KUKA KRL program: EPS_2_25618_SANMH07_A_20250918115512.src

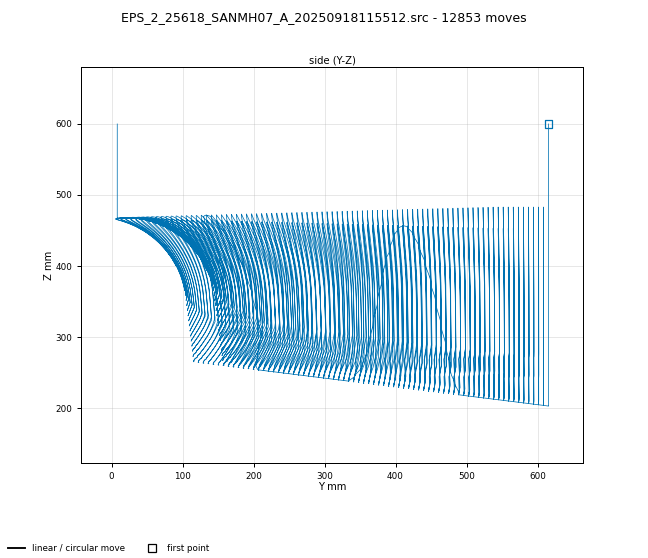
[picture p0: tool path of EPS_2_25618_SANMH07_A_20250918115512.src, 12853 of 12855 moves have a stored position in this frame; points joined in program order, loops and branches not executed]
&ACCESS RVP
&REL 4
&COMMENT QRS 19112012
&PARAM EDITMASK = *
DEF PART()
EXT BAS (BAS_COMMAND :IN,REAL :IN )
INT I
BAS (#INITMOV,0 )

;KUKA QRS Post kuka4.cps  Date:22-06-2017 !

File_ID=2844

QRS_PRE_INIT()

;Init var - Until changes are made in qrs_pre_init
Outlet_Square_prg=0
Inlet_1_Square_prg=0
Inlet_2_Square_prg=0
Inlet_3_Square_prg=0
Inlet_4_Square_prg=0
Inlet_5_Square_prg=0

Outlet_1={X 0.000, Y 540.910, Z 382.500, B 0.000, E1 0.000 }
Inlet_1={X 0.000, Y 543.050, Z 352.500, B 0.000, E1 174.000 }
Outlet_1_type=201
Inlet_1_type=201
;QRS#1=Sidecore dimensions
;QRS#2=200-8" PVC SDR 35
;QRS#3=200-8" PVC SDR 35
;QRS#4=
;QRS#5=
;QRS#6=
;QRS#7=
;QRS#8=
;QRS#9=12-08 PSX
;QRS#10=12-08 PSX
;QRS#11=
;QRS#12=
;QRS#13=
;QRS#14=
;QRS#15=
;QRS#16=1220x127x762 2,5'
;QRS#17=EPS Height
;QRS#18=483
;QRS#19=*
;QRS#20= UPDATED VERSION 22-06-2017
;QRS#21=*
Outlet_Square=0100
Inlet_1_Square=0100
Inlet_2_Square=0
Inlet_3_Square=0
Inlet_4_Square=0
Inlet_5_Square=0
Mill_Square=1
Outlet_Square_Prg=204
Inlet_1_Square_prg=204

QRS_INIT()

$ADVANCE=5

; T1
PTP {E1 173.635,E2 173.635}
PTP {X 0,Y 615.464,A -85,B 0,C 180,E1 173.635,E2 173.635,E3 0,E4 0,E5 0,E6 0}
QRS_SPEED_INIT()
LIN {X 0,Y 615.464,Z 600,A -85,B 0,C 180,E1 173.635,E2 173.635,E3 0,E4 0,E5 0,E6 0} C_VEL
LIN {X 0,Y 615.464,Z 212.869,A -85,B 0,C 180,E1 173.635,E2 173.635} C_VEL
LIN {X 0,Y 615.464,Z 204.689,A -85,B 0,C 180,E1 173.635,E2 173.635} C_VEL
LIN {X 0,Y 615.455,Z 202.689,A -85,B 0,C 180,E1 173.448,E2 173.448} C_VEL
LIN {X 0,Y 615.475,Z 202.697,A -85,B 0,C 180,E1 170.801,E2 170.801} C_VEL
LIN {X 0,Y 615.493,Z 202.687,A -85,B 0,C 180,E1 168.139,E2 168.139} C_VEL
LIN {X 0,Y 615.456,Z 202.689,A -85,B 0,C 180,E1 165.45,E2 165.45} C_VEL
LIN {X 0,Y 615.483,Z 202.698,A -85,B 0,C 180,E1 162.729,E2 162.729} C_VEL
LIN {X 0,Y 615.487,Z 202.685,A -85,B 0,C 180,E1 159.967,E2 159.967} C_VEL
LIN {X 0,Y 615.466,Z 202.687,A -85,B 0,C 180,E1 157.659,E2 157.659} C_VEL
LIN {X 0,Y 615.461,Z 202.695,A -85,B 0,C 180,E1 155.007,E2 155.007} C_VEL
LIN {X 0,Y 615.488,Z 202.687,A -85,B 0,C 180,E1 152.085,E2 152.085} C_VEL
LIN {X 0,Y 615.482,Z 202.684,A -85,B 0,C 180,E1 149.839,E2 149.839} C_VEL
LIN {X 0,Y 615.46,Z 202.688,A -85,B 0,C 180,E1 147.541,E2 147.541} C_VEL
LIN {X 0,Y 615.455,Z 202.693,A -85,B 0,C 180,E1 145.183,E2 145.183} C_VEL
LIN {X 0,Y 615.48,Z 202.698,A -85,B 0,C 180,E1 142.757,E2 142.757} C_VEL
LIN {X 0,Y 615.489,Z 202.683,A -85,B 0,C 180,E1 139.911,E2 139.911} C_VEL
LIN {X 0,Y 615.466,Z 202.687,A -85,B 0,C 180,E1 137.645,E2 137.645} C_VEL
LIN {X 0,Y 615.468,Z 202.696,A -85,B 0,C 180,E1 134.929,E2 134.929} C_VEL
LIN {X 0,Y 615.493,Z 202.685,A -85,B 0,C 180,E1 132.08,E2 132.08} C_VEL
LIN {X 0,Y 615.473,Z 202.686,A -85,B 0,C 180,E1 129.751,E2 129.751} C_VEL
LIN {X 0,Y 615.468,Z 202.696,A -85,B 0,C 180,E1 126.934,E2 126.934} C_VEL
LIN {X 0,Y 615.491,Z 202.684,A -85,B 0,C 180,E1 124.022,E2 124.022} C_VEL
LIN {X 0,Y 615.469,Z 202.686,A -85,B 0,C 180,E1 121.687,E2 121.687} C_VEL
LIN {X 0,Y 615.456,Z 202.69,A -85,B 0,C 180,E1 119.408,E2 119.408} C_VEL
LIN {X 0,Y 615.462,Z 202.695,A -85,B 0,C 180,E1 117.04,E2 117.04} C_VEL
LIN {X 0,Y 615.456,Z 202.755,A -85,B 0,C 180,E1 115.207,E2 115.207} C_VEL
LIN {X 0,Y 615.498,Z 218.624,A -85,B 0,C 180,E1 112.595,E2 112.595} C_VEL
LIN {X 0,Y 615.47,Z 236.565,A -85,B 0,C 180,E1 109.686,E2 109.686} C_VEL
LIN {X 0,Y 615.48,Z 241.935,A -85,B 0,C 180,E1 108.819,E2 108.819} C_VEL
LIN {X 0,Y 615.461,Z 349.735,A -85,B 0,C 180,E1 107.528,E2 107.528} C_VEL
LIN {X 0,Y 615.458,Z 362.991,A -85,B 0,C 180,E1 107.229,E2 107.229} C_VEL
LIN {X 0,Y 615.483,Z 375.732,A -85,B 0,C 180,E1 106.8,E2 106.8} C_VEL
LIN {X 0,Y 615.49,Z 388.024,A -85,B 0,C 180,E1 106.233,E2 106.233} C_VEL
LIN {X 0,Y 615.491,Z 399.312,A -85,B 0,C 180,E1 105.565,E2 105.565} C_VEL
LIN {X 0,Y 615.499,Z 409.63,A -85,B 0,C 180,E1 104.802,E2 104.802} C_VEL
LIN {X 0,Y 615.497,Z 419.666,A -85,B 0,C 180,E1 103.874,E2 103.874} C_VEL
LIN {X 0,Y 615.496,Z 427.092,A -85,B 0,C 180,E1 103.033,E2 103.033} C_VEL
LIN {X 0,Y 615.499,Z 434.353,A -85,B 0,C 180,E1 102.028,E2 102.028} C_VEL
LIN {X 0,Y 615.494,Z 440.767,A -85,B 0,C 180,E1 100.89,E2 100.89} C_VEL
LIN {X 0,Y 615.497,Z 445.221,A -85,B 0,C 180,E1 99.862,E2 99.862} C_VEL
LIN {X 0,Y 615.497,Z 447.492,A -85,B 0,C 180,E1 99.199,E2 99.199} C_VEL
LIN {X 0,Y 615.494,Z 449.322,A -85,B 0,C 180,E1 98.537,E2 98.537} C_VEL
LIN {X 0,Y 615.497,Z 450.679,A -85,B 0,C 180,E1 97.876,E2 97.876} C_VEL
LIN {X 0,Y 615.495,Z 452.211,A -85,B 0,C 180,E1 96.557,E2 96.557} C_VEL
LIN {X 0,Y 615.497,Z 452.381,A -85,B 0,C 180,E1 95.898,E2 95.898} C_VEL
LIN {X 0,Y 615.496,Z 451.507,A -85,B 0,C 180,E1 94.585,E2 94.585} C_VEL
LIN {X 0,Y 615.496,Z 450.503,A -85,B 0,C 180,E1 93.928,E2 93.928} C_VEL
LIN {X 0,Y 615.495,Z 449.063,A -85,B 0,C 180,E1 93.273,E2 93.273} C_VEL
LIN {X 0,Y 615.498,Z 446.127,A -85,B 0,C 180,E1 92.29,E2 92.29} C_VEL
LIN {X 0,Y 615.497,Z 442.167,A -85,B 0,C 180,E1 91.309,E2 91.309} C_VEL
LIN {X 0,Y 615.495,Z 437.073,A -85,B 0,C 180,E1 90.327,E2 90.327} C_VEL
LIN {X 0,Y 615.496,Z 430.676,A -85,B 0,C 180,E1 89.346,E2 89.346} C_VEL
LIN {X 0,Y 615.498,Z 422.726,A -85,B 0,C 180,E1 88.364,E2 88.364} C_VEL
LIN {X 0,Y 615.497,Z 414.64,A -85,B 0,C 180,E1 87.546,E2 87.546} C_VEL
LIN {X 0,Y 615.498,Z 404.769,A -85,B 0,C 180,E1 86.727,E2 86.727} C_VEL
LIN {X 0,Y 615.493,Z 393.637,A -85,B 0,C 180,E1 85.99,E2 85.99} C_VEL
LIN {X 0,Y 615.49,Z 382.757,A -85,B 0,C 180,E1 85.415,E2 85.415} C_VEL
LIN {X 0,Y 615.474,Z 370.723,A -85,B 0,C 180,E1 84.923,E2 84.923} C_VEL
LIN {X 0,Y 615.466,Z 358.081,A -85,B 0,C 180,E1 84.553,E2 84.553} C_VEL
LIN {X 0,Y 615.474,Z 344.763,A -85,B 0,C 180,E1 84.307,E2 84.307} C_VEL
LIN {X 0,Y 615.484,Z 241.899,A -85,B 0,C 180,E1 83.085,E2 83.085} C_VEL
LIN {X 0,Y 615.473,Z 224.7,A -85,B 0,C 180,E1 80.304,E2 80.304} C_VEL
LIN {X 0,Y 615.491,Z 207.383,A -85,B 0,C 180,E1 77.47,E2 77.47} C_VEL
LIN {X 0,Y 615.461,Z 202.691,A -85,B 0,C 180,E1 76.672,E2 76.672} C_VEL
LIN {X 0,Y 615.484,Z 202.683,A -85,B 0,C 180,E1 74.095,E2 74.095} C_VEL
LIN {X 0,Y 615.488,Z 202.701,A -85,B 0,C 180,E1 71.354,E2 71.354} C_VEL
LIN {X 0,Y 615.461,Z 202.689,A -85,B 0,C 180,E1 68.567,E2 68.567} C_VEL
LIN {X 0,Y 615.488,Z 202.689,A -85,B 0,C 180,E1 65.728,E2 65.728} C_VEL
LIN {X 0,Y 615.463,Z 202.693,A -85,B 0,C 180,E1 62.822,E2 62.822} C_VEL
LIN {X 0,Y 615.479,Z 202.684,A -85,B 0,C 180,E1 60.207,E2 60.207} C_VEL
LIN {X 0,Y 615.491,Z 202.694,A -85,B 0,C 180,E1 57.543,E2 57.543} C_VEL
LIN {X 0,Y 615.485,Z 202.698,A -85,B 0,C 180,E1 55.185,E2 55.185} C_VEL
LIN {X 0,Y 615.458,Z 202.692,A -85,B 0,C 180,E1 52.756,E2 52.756} C_VEL
LIN {X 0,Y 615.495,Z 202.684,A -85,B 0,C 180,E1 49.911,E2 49.911} C_VEL
LIN {X 0,Y 615.467,Z 202.695,A -85,B 0,C 180,E1 46.955,E2 46.955} C_VEL
LIN {X 0,Y 615.484,Z 202.683,A -85,B 0,C 180,E1 44.15,E2 44.15} C_VEL
LIN {X 0,Y 615.49,Z 202.697,A -85,B 0,C 180,E1 41.474,E2 41.474} C_VEL
LIN {X 0,Y 615.463,Z 202.694,A -85,B 0,C 180,E1 38.906,E2 38.906} C_VEL
LIN {X 0,Y 615.464,Z 202.687,A -85,B 0,C 180,E1 36.427,E2 36.427} C_VEL
LIN {X 0,Y 615.492,Z 202.695,A -85,B 0,C 180,E1 33.535,E2 33.535} C_VEL
LIN {X 0,Y 615.463,Z 202.694,A -85,B 0,C 180,E1 30.921,E2 30.921} C_VEL
LIN {X 0,Y 615.462,Z 202.688,A -85,B 0,C 180,E1 28.446,E2 28.446} C_VEL
LIN {X 0,Y 615.492,Z 202.694,A -85,B 0,C 180,E1 25.57,E2 25.57} C_VEL
LIN {X 0,Y 615.458,Z 202.693,A -85,B 0,C 180,E1 22.846,E2 22.846} C_VEL
LIN {X 0,Y 615.458,Z 202.689,A -85,B 0,C 180,E1 20.55,E2 20.55} C_VEL
LIN {X 0,Y 615.493,Z 202.684,A -85,B 0,C 180,E1 17.957,E2 17.957} C_VEL
LIN {X 0,Y 615.478,Z 202.699,A -85,B 0,C 180,E1 15.226,E2 15.226} C_VEL
LIN {X 0,Y 615.457,Z 202.689,A -85,B 0,C 180,E1 12.531,E2 12.531} C_VEL
LIN {X 0,Y 615.492,Z 202.686,A -85,B 0,C 180,E1 9.862,E2 9.862} C_VEL
LIN {X 0,Y 615.478,Z 202.699,A -85,B 0,C 180,E1 7.216,E2 7.216} C_VEL
LIN {X 0,Y 615.457,Z 202.69,A -85,B 0,C 180,E1 4.585,E2 4.585} C_VEL
LIN {X 0,Y 615.497,Z 202.683,A -85,B 0,C 180,E1 1.963,E2 1.963} C_VEL
LIN {X 0,Y 615.485,Z 202.702,A -85,B 0,C 180,E1 -0.654,E2 -0.654} C_VEL
LIN {X 0,Y 615.455,Z 202.692,A -85,B 0,C 180,E1 -3.273,E2 -3.273} C_VEL
LIN {X 0,Y 615.487,Z 202.684,A -85,B 0,C 180,E1 -5.899,E2 -5.899} C_VEL
LIN {X 0,Y 615.493,Z 202.699,A -85,B 0,C 180,E1 -8.537,E2 -8.537} C_VEL
LIN {X 0,Y 615.455,Z 202.693,A -85,B 0,C 180,E1 -11.194,E2 -11.194} C_VEL
LIN {X 0,Y 615.492,Z 202.683,A -85,B 0,C 180,E1 -13.934,E2 -13.934} C_VEL
LIN {X 0,Y 615.489,Z 202.702,A -85,B 0,C 180,E1 -16.587,E2 -16.587} C_VEL
LIN {X 0,Y 615.452,Z 202.691,A -85,B 0,C 180,E1 -19.339,E2 -19.339} C_VEL
LIN {X 0,Y 615.494,Z 202.687,A -85,B 0,C 180,E1 -22.136,E2 -22.136} C_VEL
LIN {X 0,Y 615.461,Z 202.695,A -85,B 0,C 180,E1 -24.993,E2 -24.993} C_VEL
LIN {X 0,Y 615.454,Z 202.693,A -85,B 0,C 180,E1 -27.179,E2 -27.179} C_VEL
LIN {X 0,Y 615.477,Z 202.685,A -85,B 0,C 180,E1 -29.793,E2 -29.793} C_VEL
LIN {X 0,Y 615.489,Z 202.698,A -85,B 0,C 180,E1 -32.457,E2 -32.457} C_VEL
LIN {X 0,Y 615.472,Z 202.697,A -85,B 0,C 180,E1 -34.816,E2 -34.816} C_VEL
LIN {X 0,Y 615.452,Z 202.692,A -85,B 0,C 180,E1 -37.245,E2 -37.245} C_VEL
LIN {X 0,Y 615.496,Z 202.686,A -85,B 0,C 180,E1 -40.09,E2 -40.09} C_VEL
LIN {X 0,Y 615.493,Z 202.694,A -85,B 0,C 180,E1 -42.353,E2 -42.353} C_VEL
LIN {X 0,Y 615.454,Z 202.694,A -85,B 0,C 180,E1 -45.072,E2 -45.072} C_VEL
LIN {X 0,Y 615.486,Z 202.685,A -85,B 0,C 180,E1 -47.92,E2 -47.92} C_VEL
LIN {X 0,Y 615.49,Z 202.692,A -85,B 0,C 180,E1 -50.25,E2 -50.25} C_VEL
LIN {X 0,Y 615.454,Z 202.694,A -85,B 0,C 180,E1 -53.068,E2 -53.068} C_VEL
LIN {X 0,Y 615.45,Z 202.691,A -85,B 0,C 180,E1 -55.305,E2 -55.305} C_VEL
LIN {X 0,Y 615.463,Z 202.688,A -85,B 0,C 180,E1 -57.673,E2 -57.673} C_VEL
LIN {X 0,Y 615.491,Z 202.7,A -85,B 0,C 180,E1 -60.594,E2 -60.594} C_VEL
LIN {X 0,Y 615.458,Z 202.695,A -85,B 0,C 180,E1 -62.961,E2 -62.961} C_VEL
LIN {X 0,Y 615.456,Z 202.695,A -85,B 0,C 180,E1 -65.007,E2 -65.007} C_VEL
LIN {X 0,Y 615.464,Z 202.688,A -85,B 0,C 180,E1 -67.66,E2 -67.66} C_VEL
LIN {X 0,Y 615.48,Z 202.765,A -85,B 0,C 180,E1 -67.838,E2 -67.838} C_VEL
LIN {X 0,Y 615.467,Z 223.077,A -85,B 0,C 180,E1 -70.661,E2 -70.661} C_VEL
LIN {X 0,Y 615.458,Z 241.931,A -85,B 0,C 180,E1 -73.242,E2 -73.242} C_VEL
LIN {X 0,Y 615.495,Z 263.271,A -85,B 0,C 180,E1 -76.126,E2 -76.126} C_VEL
LIN {X 0,Y 615.46,Z 270.645,A -85,B 0,C 180,E1 -77.113,E2 -77.113} C_VEL
LIN {X 0,Y 615.467,Z 378.836,A -85,B 0,C 180,E1 -78.41,E2 -78.41} C_VEL
LIN {X 0,Y 615.463,Z 391.349,A -85,B 0,C 180,E1 -78.681,E2 -78.681} C_VEL
LIN {X 0,Y 615.484,Z 404.665,A -85,B 0,C 180,E1 -79.115,E2 -79.115} C_VEL
LIN {X 0,Y 615.486,Z 416.478,A -85,B 0,C 180,E1 -79.639,E2 -79.639} C_VEL
LIN {X 0,Y 615.492,Z 427.995,A -85,B 0,C 180,E1 -80.304,E2 -80.304} C_VEL
LIN {X 0,Y 615.499,Z 438.341,A -85,B 0,C 180,E1 -81.05,E2 -81.05} C_VEL
LIN {X 0,Y 615.497,Z 446.812,A -85,B 0,C 180,E1 -81.794,E2 -81.794} C_VEL
LIN {X 0,Y 615.498,Z 454.606,A -85,B 0,C 180,E1 -82.62,E2 -82.62} C_VEL
LIN {X 0,Y 615.496,Z 462.203,A -85,B 0,C 180,E1 -83.608,E2 -83.608} C_VEL
LIN {X 0,Y 615.498,Z 469.205,A -85,B 0,C 180,E1 -84.759,E2 -84.759} C_VEL
LIN {X 0,Y 615.494,Z 473.851,A -85,B 0,C 180,E1 -85.744,E2 -85.744} C_VEL
LIN {X 0,Y 615.494,Z 477.399,A -85,B 0,C 180,E1 -86.727,E2 -86.727} C_VEL
LIN {X 0,Y 615.497,Z 479.233,A -85,B 0,C 180,E1 -87.382,E2 -87.382} C_VEL
LIN {X 0,Y 615.499,Z 480.608,A -85,B 0,C 180,E1 -88.037,E2 -88.037} C_VEL
LIN {X 0,Y 615.496,Z 482.173,A -85,B 0,C 180,E1 -89.346,E2 -89.346} C_VEL
LIN {X 0,Y 615.494,Z 482.389,A -85,B 0,C 180,E1 -90,E2 -90} C_VEL
LIN {X 0,Y 615.495,Z 481.58,A -85,B 0,C 180,E1 -91.309,E2 -91.309} C_VEL
LIN {X 0,Y 615.499,Z 480.608,A -85,B 0,C 180,E1 -91.963,E2 -91.963} C_VEL
LIN {X 0,Y 615.497,Z 479.233,A -85,B 0,C 180,E1 -92.618,E2 -92.618} C_VEL
LIN {X 0,Y 615.496,Z 476.349,A -85,B 0,C 180,E1 -93.601,E2 -93.601} C_VEL
LIN {X 0,Y 615.498,Z 472.441,A -85,B 0,C 180,E1 -94.584,E2 -94.584} C_VEL
LIN {X 0,Y 615.499,Z 467.405,A -85,B 0,C 180,E1 -95.57,E2 -95.57} C_VEL
LIN {X 0,Y 615.497,Z 460.869,A -85,B 0,C 180,E1 -96.583,E2 -96.583} C_VEL
LIN {X 0,Y 615.497,Z 453.133,A -85,B 0,C 180,E1 -97.545,E2 -97.545} C_VEL
LIN {X 0,Y 615.498,Z 445.045,A -85,B 0,C 180,E1 -98.371,E2 -98.371} C_VEL
LIN {X 0,Y 615.499,Z 435.167,A -85,B 0,C 180,E1 -99.199,E2 -99.199} C_VEL
LIN {X 0,Y 615.491,Z 423.98,A -85,B 0,C 180,E1 -99.945,E2 -99.945} C_VEL
LIN {X 0,Y 615.487,Z 413.022,A -85,B 0,C 180,E1 -100.527,E2 -100.527} C_VEL
LIN {X 0,Y 615.473,Z 400.516,A -85,B 0,C 180,E1 -101.039,E2 -101.039} C_VEL
LIN {X 0,Y 615.463,Z 388.069,A -85,B 0,C 180,E1 -101.402,E2 -101.402} C_VEL
LIN {X 0,Y 615.47,Z 374.468,A -85,B 0,C 180,E1 -101.652,E2 -101.652} C_VEL
LIN {X 0,Y 615.46,Z 270.645,A -85,B 0,C 180,E1 -102.887,E2 -102.887} C_VEL
LIN {X 0,Y 615.465,Z 250.722,A -85,B 0,C 180,E1 -105.566,E2 -105.566} C_VEL
LIN {X 0,Y 615.484,Z 229.594,A -85,B 0,C 180,E1 -108.442,E2 -108.442} C_VEL
LIN {X 0,Y 615.476,Z 209.239,A -85,B 0,C 180,E1 -111.257,E2 -111.257} C_VEL
LIN {X 0,Y 615.478,Z 202.686,A -85,B 0,C 180,E1 -112.187,E2 -112.187} C_VEL
LIN {X 0,Y 615.47,Z 202.687,A -85,B 0,C 180,E1 -114.273,E2 -114.273} C_VEL
LIN {X 0,Y 615.457,Z 202.689,A -85,B 0,C 180,E1 -116.446,E2 -116.446} C_VEL
LIN {X 0,Y 615.45,Z 202.691,A -85,B 0,C 180,E1 -118.66,E2 -118.66} C_VEL
LIN {X 0,Y 615.461,Z 202.696,A -85,B 0,C 180,E1 -121.081,E2 -121.081} C_VEL
LIN {X 0,Y 615.492,Z 202.685,A -85,B 0,C 180,E1 -124.022,E2 -124.022} C_VEL
LIN {X 0,Y 615.459,Z 202.688,A -85,B 0,C 180,E1 -126.427,E2 -126.427} C_VEL
LIN {X 0,Y 615.46,Z 202.695,A -85,B 0,C 180,E1 -129.059,E2 -129.059} C_VEL
LIN {X 0,Y 615.496,Z 202.701,A -85,B 0,C 180,E1 -131.473,E2 -131.473} C_VEL
LIN {X 0,Y 615.482,Z 202.685,A -85,B 0,C 180,E1 -134.15,E2 -134.15} C_VEL
LIN {X 0,Y 615.449,Z 202.692,A -85,B 0,C 180,E1 -136.752,E2 -136.752} C_VEL
LIN {X 0,Y 615.489,Z 202.7,A -85,B 0,C 180,E1 -139.394,E2 -139.394} C_VEL
LIN {X 0,Y 615.483,Z 202.688,A -85,B 0,C 180,E1 -141.989,E2 -141.989} C_VEL
LIN {X 0,Y 615.462,Z 202.688,A -85,B 0,C 180,E1 -144.382,E2 -144.382} C_VEL
LIN {X 0,Y 615.451,Z 202.692,A -85,B 0,C 180,E1 -146.761,E2 -146.761} C_VEL
LIN {X 0,Y 615.463,Z 202.696,A -85,B 0,C 180,E1 -149.079,E2 -149.079} C_VEL
LIN {X 0,Y 615.493,Z 202.698,A -85,B 0,C 180,E1 -151.549,E2 -151.549} C_VEL
LIN {X 0,Y 615.459,Z 202.688,A -85,B 0,C 180,E1 -154.437,E2 -154.437} C_VEL
LIN {X 0,Y 615.459,Z 202.688,A -85,B 0,C 180,E1 -156.442,E2 -156.442} C_VEL
LIN {X 0,Y 615.454,Z 202.69,A -85,B 0,C 180,E1 -158.567,E2 -158.567} C_VEL
LIN {X 0,Y 615.489,Z 202.699,A -85,B 0,C 180,E1 -161.354,E2 -161.354} C_VEL
LIN {X 0,Y 615.483,Z 202.685,A -85,B 0,C 180,E1 -164.095,E2 -164.095} C_VEL
LIN {X 0,Y 615.452,Z 202.692,A -85,B 0,C 180,E1 -166.798,E2 -166.798} C_VEL
LIN {X 0,Y 615.49,Z 202.701,A -85,B 0,C 180,E1 -169.473,E2 -169.473} C_VEL
LIN {X 0,Y 615.483,Z 202.685,A -85,B 0,C 180,E1 -172.124,E2 -172.124} C_VEL
LIN {X 0,Y 615.452,Z 202.692,A -85,B 0,C 180,E1 -174.759,E2 -174.759} C_VEL
LIN {X 0,Y 615.493,Z 202.7,A -85,B 0,C 180,E1 -177.382,E2 -177.382} C_VEL
LIN {X 0,Y 615.486,Z 202.686,A -85,B 0,C 180,E1 -180,E2 -180} C_VEL
LIN {X 0,Y 615.453,Z 202.69,A -85,B 0,C 180,E1 -182.618,E2 -182.618} C_VEL
LIN {X 0,Y 615.479,Z 202.698,A -85,B 0,C 180,E1 -185.241,E2 -185.241} C_VEL
LIN {X 0,Y 615.455,Z 202.689,A -85,B 0,C 180,E1 -186.552,E2 -186.552} C_VEL
LIN {X 0,Y 614.792,Z 202.845,A -85,B 0,C 180,E1 -187.098,E2 -187.098} C_VEL
LIN {X 0,Y 611.967,Z 203.251,A -85,B 0,C 180,E1 -187.984,E2 -187.984} C_VEL
LIN {X 0,Y 609.578,Z 203.566,A -85,B 0,C 180,E1 -188.696,E2 -188.696} C_VEL
LIN {X 0,Y 608.544,Z 203.686,A -85,B 0,C 180,E1 -189.246,E2 -189.246} C_VEL
LIN {X 0,Y 608.455,Z 203.693,A -85,B 0,C 180,E1 -189.432,E2 -189.432} C_VEL
LIN {X 0,Y 608.461,Z 203.688,A -85,B 0,C 180,E1 -192,E2 -192} C_VEL
LIN {X 0,Y 608.425,Z 203.691,A -85,B 0,C 180,E1 -194.722,E2 -194.722} C_VEL
LIN {X 0,Y 608.453,Z 203.697,A -85,B 0,C 180,E1 -197.477,E2 -197.477} C_VEL
LIN {X 0,Y 608.448,Z 203.688,A -85,B 0,C 180,E1 -200.275,E2 -200.275} C_VEL
LIN {X 0,Y 608.43,Z 203.69,A -85,B 0,C 180,E1 -202.47,E2 -202.47} C_VEL
LIN {X 0,Y 608.438,Z 203.689,A -85,B 0,C 180,E1 -204.572,E2 -204.572} C_VEL
LIN {X 0,Y 608.469,Z 203.692,A -85,B 0,C 180,E1 -207.205,E2 -207.205} C_VEL
LIN {X 0,Y 608.47,Z 203.687,A -85,B 0,C 180,E1 -209.972,E2 -209.972} C_VEL
LIN {X 0,Y 608.446,Z 203.69,A -85,B 0,C 180,E1 -212.88,E2 -212.88} C_VEL
LIN {X 0,Y 608.436,Z 203.698,A -85,B 0,C 180,E1 -215.278,E2 -215.278} C_VEL
LIN {X 0,Y 608.462,Z 203.686,A -85,B 0,C 180,E1 -218.24,E2 -218.24} C_VEL
LIN {X 0,Y 608.461,Z 203.696,A -85,B 0,C 180,E1 -221.342,E2 -221.342} C_VEL
LIN {X 0,Y 608.451,Z 203.687,A -85,B 0,C 180,E1 -224.263,E2 -224.263} C_VEL
LIN {X 0,Y 608.432,Z 203.694,A -85,B 0,C 180,E1 -227.038,E2 -227.038} C_VEL
LIN {X 0,Y 608.458,Z 203.692,A -85,B 0,C 180,E1 -229.697,E2 -229.697} C_VEL
LIN {X 0,Y 608.459,Z 203.686,A -85,B 0,C 180,E1 -232.253,E2 -232.253} C_VEL
LIN {X 0,Y 608.438,Z 203.695,A -85,B 0,C 180,E1 -235.097,E2 -235.097} C_VEL
LIN {X 0,Y 608.464,Z 203.688,A -85,B 0,C 180,E1 -237.905,E2 -237.905} C_VEL
LIN {X 0,Y 608.463,Z 203.686,A -85,B 0,C 180,E1 -240.22,E2 -240.22} C_VEL
LIN {X 0,Y 608.437,Z 203.691,A -85,B 0,C 180,E1 -242.801,E2 -242.801} C_VEL
LIN {X 0,Y 608.459,Z 203.892,A -85,B 0,C 180,E1 -244.745,E2 -244.745} C_VEL
LIN {X 0,Y 608.501,Z 220.588,A -85,B 0,C 180,E1 -247.515,E2 -247.515} C_VEL
LIN {X 0,Y 608.442,Z 238.425,A -85,B 0,C 180,E1 -250.429,E2 -250.429} C_VEL
LIN {X 0,Y 608.492,Z 242.41,A -85,B 0,C 180,E1 -251.044,E2 -251.044} C_VEL
LIN {X 0,Y 608.511,Z 349.433,A -85,B 0,C 180,E1 -252.33,E2 -252.33} C_VEL
LIN {X 0,Y 608.502,Z 362.826,A -85,B 0,C 180,E1 -252.633,E2 -252.633} C_VEL
LIN {X 0,Y 608.516,Z 375.098,A -85,B 0,C 180,E1 -253.045,E2 -253.045} C_VEL
LIN {X 0,Y 608.511,Z 386.902,A -85,B 0,C 180,E1 -253.578,E2 -253.578} C_VEL
LIN {X 0,Y 608.497,Z 398.424,A -85,B 0,C 180,E1 -254.251,E2 -254.251} C_VEL
LIN {X 0,Y 608.478,Z 409,A -85,B 0,C 180,E1 -255.023,E2 -255.023} C_VEL
LIN {X 0,Y 608.465,Z 417.618,A -85,B 0,C 180,E1 -255.792,E2 -255.792} C_VEL
LIN {X 0,Y 608.452,Z 426.884,A -85,B 0,C 180,E1 -256.813,E2 -256.813} C_VEL
LIN {X 0,Y 608.44,Z 434.314,A -85,B 0,C 180,E1 -257.831,E2 -257.831} C_VEL
LIN {X 0,Y 608.459,Z 440.697,A -85,B 0,C 180,E1 -258.938,E2 -258.938} C_VEL
LIN {X 0,Y 608.437,Z 445.495,A -85,B 0,C 180,E1 -260.022,E2 -260.022} C_VEL
LIN {X 0,Y 608.426,Z 447.826,A -85,B 0,C 180,E1 -260.693,E2 -260.693} C_VEL
LIN {X 0,Y 608.421,Z 449.722,A -85,B 0,C 180,E1 -261.363,E2 -261.363} C_VEL
LIN {X 0,Y 608.423,Z 451.157,A -85,B 0,C 180,E1 -262.032,E2 -262.032} C_VEL
LIN {X 0,Y 608.448,Z 452.772,A -85,B 0,C 180,E1 -263.367,E2 -263.367} C_VEL
LIN {X 0,Y 608.434,Z 453,A -85,B 0,C 180,E1 -264.033,E2 -264.033} C_VEL
LIN {X 0,Y 608.429,Z 452.192,A -85,B 0,C 180,E1 -265.362,E2 -265.362} C_VEL
LIN {X 0,Y 608.433,Z 451.21,A -85,B 0,C 180,E1 -266.026,E2 -266.026} C_VEL
LIN {X 0,Y 608.424,Z 449.82,A -85,B 0,C 180,E1 -266.689,E2 -266.689} C_VEL
LIN {X 0,Y 608.43,Z 446.911,A -85,B 0,C 180,E1 -267.683,E2 -267.683} C_VEL
LIN {X 0,Y 608.45,Z 442.978,A -85,B 0,C 180,E1 -268.676,E2 -268.676} C_VEL
LIN {X 0,Y 608.441,Z 437.923,A -85,B 0,C 180,E1 -269.669,E2 -269.669} C_VEL
LIN {X 0,Y 608.442,Z 431.589,A -85,B 0,C 180,E1 -270.662,E2 -270.662} C_VEL
LIN {X 0,Y 608.464,Z 423.686,A -85,B 0,C 180,E1 -271.655,E2 -271.655} C_VEL
LIN {X 0,Y 608.49,Z 413.901,A -85,B 0,C 180,E1 -272.648,E2 -272.648} C_VEL
LIN {X 0,Y 608.478,Z 403.672,A -85,B 0,C 180,E1 -273.476,E2 -273.476} C_VEL
LIN {X 0,Y 608.501,Z 392.204,A -85,B 0,C 180,E1 -274.222,E2 -274.222} C_VEL
LIN {X 0,Y 608.532,Z 380.856,A -85,B 0,C 180,E1 -274.803,E2 -274.803} C_VEL
LIN {X 0,Y 608.498,Z 367.931,A -85,B 0,C 180,E1 -275.302,E2 -275.302} C_VEL
LIN {X 0,Y 608.531,Z 354.902,A -85,B 0,C 180,E1 -275.654,E2 -275.654} C_VEL
LIN {X 0,Y 608.535,Z 342.327,A -85,B 0,C 180,E1 -275.862,E2 -275.862} C_VEL
LIN {X 0,Y 608.47,Z 242.193,A -85,B 0,C 180,E1 -277.049,E2 -277.049} C_VEL
LIN {X 0,Y 608.471,Z 225.253,A -85,B 0,C 180,E1 -279.809,E2 -279.809} C_VEL
LIN {X 0,Y 608.493,Z 208.91,A -85,B 0,C 180,E1 -282.507,E2 -282.507} C_VEL
LIN {X 0,Y 608.454,Z 203.689,A -85,B 0,C 180,E1 -283.399,E2 -283.399} C_VEL
LIN {X 0,Y 608.461,Z 203.688,A -85,B 0,C 180,E1 -286.094,E2 -286.094} C_VEL
LIN {X 0,Y 608.453,Z 203.695,A -85,B 0,C 180,E1 -288.87,E2 -288.87} C_VEL
LIN {X 0,Y 608.458,Z 203.686,A -85,B 0,C 180,E1 -291.692,E2 -291.692} C_VEL
LIN {X 0,Y 608.45,Z 203.696,A -85,B 0,C 180,E1 -294.571,E2 -294.571} C_VEL
LIN {X 0,Y 608.441,Z 203.691,A -85,B 0,C 180,E1 -297.2,E2 -297.2} C_VEL
LIN {X 0,Y 608.464,Z 203.686,A -85,B 0,C 180,E1 -299.78,E2 -299.78} C_VEL
LIN {X 0,Y 608.465,Z 203.694,A -85,B 0,C 180,E1 -302.522,E2 -302.522} C_VEL
LIN {X 0,Y 608.433,Z 203.691,A -85,B 0,C 180,E1 -305.278,E2 -305.278} C_VEL
LIN {X 0,Y 608.468,Z 203.689,A -85,B 0,C 180,E1 -308.24,E2 -308.24} C_VEL
LIN {X 0,Y 608.433,Z 203.692,A -85,B 0,C 180,E1 -311.178,E2 -311.178} C_VEL
LIN {X 0,Y 608.467,Z 203.686,A -85,B 0,C 180,E1 -313.87,E2 -313.87} C_VEL
LIN {X 0,Y 608.475,Z 203.695,A -85,B 0,C 180,E1 -316.691,E2 -316.691} C_VEL
LIN {X 0,Y 608.448,Z 203.696,A -85,B 0,C 180,E1 -318.822,E2 -318.822} C_VEL
LIN {X 0,Y 608.461,Z 203.686,A -85,B 0,C 180,E1 -321.76,E2 -321.76} C_VEL
LIN {X 0,Y 608.448,Z 203.689,A -85,B 0,C 180,E1 -323.954,E2 -323.954} C_VEL
LIN {X 0,Y 608.469,Z 203.69,A -85,B 0,C 180,E1 -326.329,E2 -326.329} C_VEL
LIN {X 0,Y 608.445,Z 203.698,A -85,B 0,C 180,E1 -328.733,E2 -328.733} C_VEL
LIN {X 0,Y 608.451,Z 203.688,A -85,B 0,C 180,E1 -331.384,E2 -331.384} C_VEL
LIN {X 0,Y 608.438,Z 203.69,A -85,B 0,C 180,E1 -333.964,E2 -333.964} C_VEL
LIN {X 0,Y 608.438,Z 203.695,A -85,B 0,C 180,E1 -336.875,E2 -336.875} C_VEL
LIN {X 0,Y 608.446,Z 203.689,A -85,B 0,C 180,E1 -339.327,E2 -339.327} C_VEL
LIN {X 0,Y 608.444,Z 203.688,A -85,B 0,C 180,E1 -341.828,E2 -341.828} C_VEL
LIN {X 0,Y 608.467,Z 203.696,A -85,B 0,C 180,E1 -344.594,E2 -344.594} C_VEL
LIN {X 0,Y 608.454,Z 203.688,A -85,B 0,C 180,E1 -347.322,E2 -347.322} C_VEL
LIN {X 0,Y 608.456,Z 203.688,A -85,B 0,C 180,E1 -350.023,E2 -350.023} C_VEL
LIN {X 0,Y 608.46,Z 203.696,A -85,B 0,C 180,E1 -352.7,E2 -352.7} C_VEL
LIN {X 0,Y 608.464,Z 203.695,A -85,B 0,C 180,E1 -354.698,E2 -354.698} C_VEL
LIN {X 0,Y 608.451,Z 203.688,A -85,B 0,C 180,E1 -357.352,E2 -357.352} C_VEL
LIN {X 0,Y 608.477,Z 203.686,A -85,B 0,C 180,E1 -360,E2 -360} C_VEL
LIN {X 0,Y 608.481,Z 203.694,A -85,B 0,C 180,E1 -362.648,E2 -362.648} C_VEL
LIN {X 0,Y 608.439,Z 203.69,A -85,B 0,C 180,E1 -365.302,E2 -365.302} C_VEL
LIN {X 0,Y 608.477,Z 203.686,A -85,B 0,C 180,E1 -367.967,E2 -367.967} C_VEL
LIN {X 0,Y 608.461,Z 203.691,A -85,B 0,C 180,E1 -370.952,E2 -370.952} C_VEL
LIN {X 0,Y 608.441,Z 203.689,A -85,B 0,C 180,E1 -373.357,E2 -373.357} C_VEL
LIN {X 0,Y 608.46,Z 203.689,A -85,B 0,C 180,E1 -376.094,E2 -376.094} C_VEL
LIN {X 0,Y 608.45,Z 203.693,A -85,B 0,C 180,E1 -378.87,E2 -378.87} C_VEL
LIN {X 0,Y 608.454,Z 203.687,A -85,B 0,C 180,E1 -381.692,E2 -381.692} C_VEL
LIN {X 0,Y 608.447,Z 203.699,A -85,B 0,C 180,E1 -384.571,E2 -384.571} C_VEL
LIN {X 0,Y 608.433,Z 203.691,A -85,B 0,C 180,E1 -387.199,E2 -387.199} C_VEL
LIN {X 0,Y 608.462,Z 203.686,A -85,B 0,C 180,E1 -389.78,E2 -389.78} C_VEL
LIN {X 0,Y 608.463,Z 203.696,A -85,B 0,C 180,E1 -392.523,E2 -392.523} C_VEL
LIN {X 0,Y 608.426,Z 203.691,A -85,B 0,C 180,E1 -395.279,E2 -395.279} C_VEL
LIN {X 0,Y 608.466,Z 203.691,A -85,B 0,C 180,E1 -398.24,E2 -398.24} C_VEL
LIN {X 0,Y 608.421,Z 203.693,A -85,B 0,C 180,E1 -401.18,E2 -401.18} C_VEL
LIN {X 0,Y 608.465,Z 203.687,A -85,B 0,C 180,E1 -403.87,E2 -403.87} C_VEL
LIN {X 0,Y 608.466,Z 203.694,A -85,B 0,C 180,E1 -406.692,E2 -406.692} C_VEL
LIN {X 0,Y 608.44,Z 203.695,A -85,B 0,C 180,E1 -408.822,E2 -408.822} C_VEL
LIN {X 0,Y 608.459,Z 203.687,A -85,B 0,C 180,E1 -411.761,E2 -411.761} C_VEL
LIN {X 0,Y 608.435,Z 203.697,A -85,B 0,C 180,E1 -414.722,E2 -414.722} C_VEL
LIN {X 0,Y 608.442,Z 203.69,A -85,B 0,C 180,E1 -417.12,E2 -417.12} C_VEL
LIN {X 0,Y 608.47,Z 203.688,A -85,B 0,C 180,E1 -420.028,E2 -420.028} C_VEL
LIN {X 0,Y 608.463,Z 203.692,A -85,B 0,C 180,E1 -422.796,E2 -422.796} C_VEL
LIN {X 0,Y 608.435,Z 203.689,A -85,B 0,C 180,E1 -425.428,E2 -425.428} C_VEL
LIN {X 0,Y 608.474,Z 203.891,A -85,B 0,C 180,E1 -427.729,E2 -427.729} C_VEL
LIN {X 0,Y 608.549,Z 220.577,A -85,B 0,C 180,E1 -430.081,E2 -430.081} C_VEL
LIN {X 0,Y 608.478,Z 240.726,A -85,B 0,C 180,E1 -432.871,E2 -432.871} C_VEL
LIN {X 0,Y 608.501,Z 260.875,A -85,B 0,C 180,E1 -435.622,E2 -435.622} C_VEL
LIN {X 0,Y 608.467,Z 271.144,A -85,B 0,C 180,E1 -436.984,E2 -436.984} C_VEL
LIN {X 0,Y 608.531,Z 378.948,A -85,B 0,C 180,E1 -438.276,E2 -438.276} C_VEL
LIN {X 0,Y 608.498,Z 392.217,A -85,B 0,C 180,E1 -438.571,E2 -438.571} C_VEL
LIN {X 0,Y 608.51,Z 404.166,A -85,B 0,C 180,E1 -438.965,E2 -438.965} C_VEL
LIN {X 0,Y 608.505,Z 416.635,A -85,B 0,C 180,E1 -439.519,E2 -439.519} C_VEL
LIN {X 0,Y 608.483,Z 428.198,A -85,B 0,C 180,E1 -440.191,E2 -440.191} C_VEL
LIN {X 0,Y 608.485,Z 438.594,A -85,B 0,C 180,E1 -440.946,E2 -440.946} C_VEL
LIN {X 0,Y 608.475,Z 447.112,A -85,B 0,C 180,E1 -441.699,E2 -441.699} C_VEL
LIN {X 0,Y 608.471,Z 454.96,A -85,B 0,C 180,E1 -442.534,E2 -442.534} C_VEL
LIN {X 0,Y 608.461,Z 462.286,A -85,B 0,C 180,E1 -443.484,E2 -443.484} C_VEL
LIN {X 0,Y 608.45,Z 467.866,A -85,B 0,C 180,E1 -444.366,E2 -444.366} C_VEL
LIN {X 0,Y 608.432,Z 472.95,A -85,B 0,C 180,E1 -445.362,E2 -445.362} C_VEL
LIN {X 0,Y 608.449,Z 476.896,A -85,B 0,C 180,E1 -446.358,E2 -446.358} C_VEL
LIN {X 0,Y 608.425,Z 479.809,A -85,B 0,C 180,E1 -447.352,E2 -447.352} C_VEL
LIN {X 0,Y 608.444,Z 481.201,A -85,B 0,C 180,E1 -448.014,E2 -448.014} C_VEL
LIN {X 0,Y 608.438,Z 482.783,A -85,B 0,C 180,E1 -449.338,E2 -449.338} C_VEL
LIN {X 0,Y 608.434,Z 483,A -85,B 0,C 180,E1 -450,E2 -450} C_VEL
LIN {X 0,Y 608.448,Z 482.184,A -85,B 0,C 180,E1 -451.324,E2 -451.324} C_VEL
LIN {X 0,Y 608.444,Z 481.201,A -85,B 0,C 180,E1 -451.986,E2 -451.986} C_VEL
LIN {X 0,Y 608.425,Z 479.809,A -85,B 0,C 180,E1 -452.648,E2 -452.648} C_VEL
LIN {X 0,Y 608.449,Z 476.896,A -85,B 0,C 180,E1 -453.642,E2 -453.642} C_VEL
LIN {X 0,Y 608.432,Z 472.95,A -85,B 0,C 180,E1 -454.638,E2 -454.638} C_VEL
LIN {X 0,Y 608.437,Z 466.876,A -85,B 0,C 180,E1 -455.801,E2 -455.801} C_VEL
LIN {X 0,Y 608.462,Z 460.235,A -85,B 0,C 180,E1 -456.799,E2 -456.799} C_VEL
LIN {X 0,Y 608.456,Z 451.989,A -85,B 0,C 180,E1 -457.8,E2 -457.8} C_VEL
LIN {X 0,Y 608.472,Z 443.536,A -85,B 0,C 180,E1 -458.636,E2 -458.636} C_VEL
LIN {X 0,Y 608.478,Z 433.091,A -85,B 0,C 180,E1 -459.473,E2 -459.473} C_VEL
LIN {X 0,Y 608.501,Z 422.755,A -85,B 0,C 180,E1 -460.145,E2 -460.145} C_VEL
LIN {X 0,Y 608.517,Z 411.6,A -85,B 0,C 180,E1 -460.724,E2 -460.724} C_VEL
LIN {X 0,Y 608.515,Z 399.9,A -85,B 0,C 180,E1 -461.192,E2 -461.192} C_VEL
LIN {X 0,Y 608.528,Z 387.265,A -85,B 0,C 180,E1 -461.555,E2 -461.555} C_VEL
LIN {X 0,Y 608.533,Z 374.599,A -85,B 0,C 180,E1 -461.787,E2 -461.787} C_VEL
LIN {X 0,Y 608.467,Z 271.14,A -85,B 0,C 180,E1 -463.017,E2 -463.017} C_VEL
LIN {X 0,Y 608.46,Z 253.319,A -85,B 0,C 180,E1 -465.406,E2 -465.406} C_VEL
LIN {X 0,Y 608.51,Z 233.17,A -85,B 0,C 180,E1 -468.17,E2 -468.17} C_VEL
LIN {X 0,Y 608.526,Z 214.438,A -85,B 0,C 180,E1 -470.78,E2 -470.78} C_VEL
LIN {X 0,Y 608.44,Z 203.691,A -85,B 0,C 180,E1 -472.317,E2 -472.317} C_VEL
LIN {X 0,Y 608.435,Z 203.69,A -85,B 0,C 180,E1 -474.572,E2 -474.572} C_VEL
LIN {X 0,Y 608.463,Z 203.692,A -85,B 0,C 180,E1 -477.204,E2 -477.204} C_VEL
LIN {X 0,Y 608.47,Z 203.688,A -85,B 0,C 180,E1 -479.972,E2 -479.972} C_VEL
LIN {X 0,Y 608.441,Z 203.69,A -85,B 0,C 180,E1 -482.881,E2 -482.881} C_VEL
LIN {X 0,Y 608.435,Z 203.697,A -85,B 0,C 180,E1 -485.278,E2 -485.278} C_VEL
LIN {X 0,Y 608.461,Z 203.687,A -85,B 0,C 180,E1 -488.239,E2 -488.239} C_VEL
LIN {X 0,Y 608.458,Z 203.695,A -85,B 0,C 180,E1 -491.342,E2 -491.342} C_VEL
LIN {X 0,Y 608.449,Z 203.688,A -85,B 0,C 180,E1 -494.263,E2 -494.263} C_VEL
LIN {X 0,Y 608.443,Z 203.689,A -85,B 0,C 180,E1 -496.694,E2 -496.694} C_VEL
LIN {X 0,Y 608.421,Z 203.692,A -85,B 0,C 180,E1 -498.82,E2 -498.82} C_VEL
LIN {X 0,Y 608.465,Z 203.691,A -85,B 0,C 180,E1 -501.76,E2 -501.76} C_VEL
LIN {X 0,Y 608.425,Z 203.691,A -85,B 0,C 180,E1 -504.721,E2 -504.721} C_VEL
LIN {X 0,Y 608.466,Z 203.696,A -85,B 0,C 180,E1 -507.477,E2 -507.477} C_VEL
LIN {X 0,Y 608.462,Z 203.686,A -85,B 0,C 180,E1 -510.22,E2 -510.22} C_VEL
LIN {X 0,Y 608.432,Z 203.691,A -85,B 0,C 180,E1 -512.801,E2 -512.801} C_VEL
LIN {X 0,Y 608.447,Z 203.699,A -85,B 0,C 180,E1 -515.429,E2 -515.429} C_VEL
LIN {X 0,Y 608.454,Z 203.687,A -85,B 0,C 180,E1 -518.308,E2 -518.308} C_VEL
LIN {X 0,Y 608.451,Z 203.693,A -85,B 0,C 180,E1 -521.13,E2 -521.13} C_VEL
LIN {X 0,Y 608.46,Z 203.689,A -85,B 0,C 180,E1 -523.906,E2 -523.906} C_VEL
LIN {X 0,Y 608.439,Z 203.689,A -85,B 0,C 180,E1 -526.643,E2 -526.643} C_VEL
LIN {X 0,Y 608.46,Z 203.695,A -85,B 0,C 180,E1 -529.35,E2 -529.35} C_VEL
LIN {X 0,Y 608.476,Z 203.686,A -85,B 0,C 180,E1 -532.033,E2 -532.033} C_VEL
LIN {X 0,Y 608.436,Z 203.69,A -85,B 0,C 180,E1 -534.698,E2 -534.698} C_VEL
LIN {X 0,Y 608.481,Z 203.693,A -85,B 0,C 180,E1 -537.352,E2 -537.352} C_VEL
LIN {X 0,Y 608.477,Z 203.686,A -85,B 0,C 180,E1 -540,E2 -540} C_VEL
LIN {X 0,Y 608.449,Z 203.688,A -85,B 0,C 180,E1 -542.648,E2 -542.648} C_VEL
LIN {X 0,Y 608.46,Z 203.695,A -85,B 0,C 180,E1 -545.302,E2 -545.302} C_VEL
LIN {X 0,Y 608.479,Z 203.686,A -85,B 0,C 180,E1 -547.967,E2 -547.967} C_VEL
LIN {X 0,Y 608.455,Z 203.693,A -85,B 0,C 180,E1 -549.432,E2 -549.432} C_VEL
LIN {X 0,Y 607.779,Z 203.774,A -85,B 0,C 180,E1 -549.985,E2 -549.985} C_VEL
LIN {X 0,Y 604.931,Z 204.128,A -85,B 0,C 180,E1 -550.882,E2 -550.882} C_VEL
LIN {X 0,Y 602.527,Z 204.433,A -85,B 0,C 180,E1 -551.603,E2 -551.603} C_VEL
LIN {X 0,Y 601.488,Z 204.556,A -85,B 0,C 180,E1 -552.16,E2 -552.16} C_VEL
LIN {X 0,Y 601.4,Z 204.565,A -85,B 0,C 180,E1 -552.348,E2 -552.348} C_VEL
LIN {X 0,Y 601.397,Z 204.568,A -85,B 0,C 180,E1 -554.898,E2 -554.898} C_VEL
LIN {X 0,Y 601.396,Z 204.572,A -85,B 0,C 180,E1 -557.689,E2 -557.689} C_VEL
LIN {X 0,Y 601.411,Z 204.564,A -85,B 0,C 180,E1 -560.523,E2 -560.523} C_VEL
LIN {X 0,Y 601.415,Z 204.575,A -85,B 0,C 180,E1 -563.411,E2 -563.411} C_VEL
LIN {X 0,Y 601.389,Z 204.567,A -85,B 0,C 180,E1 -566.365,E2 -566.365} C_VEL
LIN {X 0,Y 601.413,Z 204.566,A -85,B 0,C 180,E1 -568.785,E2 -568.785} C_VEL
LIN {X 0,Y 601.419,Z 204.574,A -85,B 0,C 180,E1 -571.454,E2 -571.454} C_VEL
LIN {X 0,Y 601.425,Z 204.563,A -85,B 0,C 180,E1 -574.119,E2 -574.119} C_VEL
LIN {X 0,Y 601.389,Z 204.567,A -85,B 0,C 180,E1 -576.584,E2 -576.584} C_VEL
LIN {X 0,Y 601.399,Z 204.572,A -85,B 0,C 180,E1 -579.128,E2 -579.128} C_VEL
LIN {X 0,Y 601.425,Z 204.567,A -85,B 0,C 180,E1 -581.765,E2 -581.765} C_VEL
LIN {X 0,Y 601.4,Z 204.566,A -85,B 0,C 180,E1 -584.533,E2 -584.533} C_VEL
LIN {X 0,Y 601.412,Z 204.575,A -85,B 0,C 180,E1 -587.41,E2 -587.41} C_VEL
LIN {X 0,Y 601.401,Z 204.567,A -85,B 0,C 180,E1 -590.004,E2 -590.004} C_VEL
LIN {X 0,Y 601.431,Z 204.563,A -85,B 0,C 180,E1 -592.619,E2 -592.619} C_VEL
LIN {X 0,Y 601.4,Z 204.571,A -85,B 0,C 180,E1 -595.067,E2 -595.067} C_VEL
LIN {X 0,Y 601.435,Z 204.571,A -85,B 0,C 180,E1 -597.484,E2 -597.484} C_VEL
LIN {X 0,Y 601.431,Z 204.565,A -85,B 0,C 180,E1 -599.852,E2 -599.852} C_VEL
LIN {X 0,Y 601.39,Z 204.568,A -85,B 0,C 180,E1 -602.643,E2 -602.643} C_VEL
LIN {X 0,Y 601.409,Z 204.64,A -85,B 0,C 180,E1 -604.636,E2 -604.636} C_VEL
LIN {X 0,Y 601.463,Z 217.338,A -85,B 0,C 180,E1 -606.774,E2 -606.774} C_VEL
LIN {X 0,Y 601.445,Z 233.634,A -85,B 0,C 180,E1 -609.479,E2 -609.479} C_VEL
LIN {X 0,Y 601.398,Z 242.152,A -85,B 0,C 180,E1 -610.878,E2 -610.878} C_VEL
LIN {X 0,Y 601.651,Z 247.159,A -85,B 0,C 180,E1 -610.951,E2 -610.951} C_VEL
LIN {X 0,Y 601.558,Z 349.016,A -85,B 0,C 180,E1 -612.185,E2 -612.185} C_VEL
LIN {X 0,Y 601.531,Z 362.545,A -85,B 0,C 180,E1 -612.491,E2 -612.491} C_VEL
LIN {X 0,Y 601.549,Z 375.47,A -85,B 0,C 180,E1 -612.93,E2 -612.93} C_VEL
LIN {X 0,Y 601.525,Z 387.146,A -85,B 0,C 180,E1 -613.469,E2 -613.469} C_VEL
LIN {X 0,Y 601.479,Z 398.634,A -85,B 0,C 180,E1 -614.15,E2 -614.15} C_VEL
LIN {X 0,Y 601.46,Z 409.176,A -85,B 0,C 180,E1 -614.931,E2 -614.931} C_VEL
LIN {X 0,Y 601.424,Z 418.592,A -85,B 0,C 180,E1 -615.795,E2 -615.795} C_VEL
LIN {X 0,Y 601.396,Z 427.688,A -85,B 0,C 180,E1 -616.828,E2 -616.828} C_VEL
LIN {X 0,Y 601.371,Z 434.958,A -85,B 0,C 180,E1 -617.857,E2 -617.857} C_VEL
LIN {X 0,Y 601.34,Z 441.438,A -85,B 0,C 180,E1 -619.032,E2 -619.032} C_VEL
LIN {X 0,Y 601.341,Z 446.484,A -85,B 0,C 180,E1 -620.243,E2 -620.243} C_VEL
LIN {X 0,Y 601.333,Z 449.535,A -85,B 0,C 180,E1 -621.261,E2 -621.261} C_VEL
LIN {X 0,Y 601.334,Z 451.036,A -85,B 0,C 180,E1 -621.938,E2 -621.938} C_VEL
LIN {X 0,Y 601.358,Z 452.724,A -85,B 0,C 180,E1 -623.289,E2 -623.289} C_VEL
LIN {X 0,Y 601.333,Z 452.987,A -85,B 0,C 180,E1 -623.962,E2 -623.962} C_VEL
LIN {X 0,Y 601.334,Z 452.839,A -85,B 0,C 180,E1 -624.635,E2 -624.635} C_VEL
LIN {X 0,Y 601.342,Z 451.325,A -85,B 0,C 180,E1 -625.979,E2 -625.979} C_VEL
LIN {X 0,Y 601.34,Z 449.982,A -85,B 0,C 180,E1 -626.65,E2 -626.65} C_VEL
LIN {X 0,Y 601.341,Z 447.134,A -85,B 0,C 180,E1 -627.656,E2 -627.656} C_VEL
LIN {X 0,Y 601.352,Z 443.276,A -85,B 0,C 180,E1 -628.661,E2 -628.661} C_VEL
LIN {X 0,Y 601.368,Z 438.302,A -85,B 0,C 180,E1 -629.665,E2 -629.665} C_VEL
LIN {X 0,Y 601.367,Z 432.075,A -85,B 0,C 180,E1 -630.67,E2 -630.67} C_VEL
LIN {X 0,Y 601.408,Z 424.307,A -85,B 0,C 180,E1 -631.674,E2 -631.674} C_VEL
LIN {X 0,Y 601.428,Z 414.647,A -85,B 0,C 180,E1 -632.679,E2 -632.679} C_VEL
LIN {X 0,Y 601.454,Z 404.639,A -85,B 0,C 180,E1 -633.517,E2 -633.517} C_VEL
LIN {X 0,Y 601.482,Z 393.379,A -85,B 0,C 180,E1 -634.272,E2 -634.272} C_VEL
LIN {X 0,Y 601.528,Z 382.353,A -85,B 0,C 180,E1 -634.859,E2 -634.859} C_VEL
LIN {X 0,Y 601.528,Z 370.072,A -85,B 0,C 180,E1 -635.363,E2 -635.363} C_VEL
LIN {X 0,Y 601.589,Z 357.015,A -85,B 0,C 180,E1 -635.741,E2 -635.741} C_VEL
LIN {X 0,Y 601.61,Z 344.436,A -85,B 0,C 180,E1 -635.972,E2 -635.972} C_VEL
LIN {X 0,Y 601.637,Z 243.619,A -85,B 0,C 180,E1 -637.182,E2 -637.182} C_VEL
LIN {X 0,Y 601.401,Z 242.122,A -85,B 0,C 180,E1 -637.217,E2 -637.217} C_VEL
LIN {X 0,Y 601.466,Z 225.693,A -85,B 0,C 180,E1 -639.924,E2 -639.924} C_VEL
LIN {X 0,Y 601.526,Z 207.316,A -85,B 0,C 180,E1 -642.998,E2 -642.998} C_VEL
LIN {X 0,Y 601.404,Z 204.568,A -85,B 0,C 180,E1 -643.473,E2 -643.473} C_VEL
LIN {X 0,Y 601.442,Z 204.565,A -85,B 0,C 180,E1 -646.287,E2 -646.287} C_VEL
LIN {X 0,Y 601.415,Z 204.568,A -85,B 0,C 180,E1 -649.099,E2 -649.099} C_VEL
LIN {X 0,Y 601.402,Z 204.568,A -85,B 0,C 180,E1 -651.239,E2 -651.239} C_VEL
LIN {X 0,Y 601.462,Z 204.56,A -85,B 0,C 180,E1 -654.14,E2 -654.14} C_VEL
LIN {X 0,Y 601.403,Z 204.569,A -85,B 0,C 180,E1 -657.113,E2 -657.113} C_VEL
LIN {X 0,Y 601.401,Z 204.566,A -85,B 0,C 180,E1 -659.394,E2 -659.394} C_VEL
LIN {X 0,Y 601.4,Z 204.566,A -85,B 0,C 180,E1 -661.727,E2 -661.727} C_VEL
LIN {X 0,Y 601.424,Z 204.565,A -85,B 0,C 180,E1 -664.119,E2 -664.119} C_VEL
LIN {X 0,Y 601.398,Z 204.575,A -85,B 0,C 180,E1 -666.583,E2 -666.583} C_VEL
LIN {X 0,Y 601.402,Z 204.569,A -85,B 0,C 180,E1 -669.127,E2 -669.127} C_VEL
LIN {X 0,Y 601.422,Z 204.563,A -85,B 0,C 180,E1 -671.765,E2 -671.765} C_VEL
LIN {X 0,Y 601.427,Z 204.571,A -85,B 0,C 180,E1 -674.535,E2 -674.535} C_VEL
LIN {X 0,Y 601.384,Z 204.569,A -85,B 0,C 180,E1 -677.327,E2 -677.327} C_VEL
LIN {X 0,Y 601.403,Z 204.566,A -85,B 0,C 180,E1 -680.004,E2 -680.004} C_VEL
LIN {X 0,Y 601.435,Z 204.572,A -85,B 0,C 180,E1 -682.618,E2 -682.618} C_VEL
LIN {X 0,Y 601.393,Z 204.57,A -85,B 0,C 180,E1 -685.066,E2 -685.066} C_VEL
LIN {X 0,Y 601.413,Z 204.564,A -85,B 0,C 180,E1 -687.483,E2 -687.483} C_VEL
LIN {X 0,Y 601.43,Z 204.562,A -85,B 0,C 180,E1 -689.851,E2 -689.851} C_VEL
LIN {X 0,Y 601.423,Z 204.569,A -85,B 0,C 180,E1 -692.887,E2 -692.887} C_VEL
LIN {X 0,Y 601.416,Z 204.564,A -85,B 0,C 180,E1 -695.712,E2 -695.712} C_VEL
LIN {X 0,Y 601.403,Z 204.567,A -85,B 0,C 180,E1 -698.04,E2 -698.04} C_VEL
LIN {X 0,Y 601.413,Z 204.57,A -85,B 0,C 180,E1 -700.901,E2 -700.901} C_VEL
LIN {X 0,Y 601.418,Z 204.563,A -85,B 0,C 180,E1 -703.712,E2 -703.712} C_VEL
LIN {X 0,Y 601.418,Z 204.572,A -85,B 0,C 180,E1 -706.484,E2 -706.484} C_VEL
LIN {X 0,Y 601.397,Z 204.568,A -85,B 0,C 180,E1 -709.223,E2 -709.223} C_VEL
LIN {X 0,Y 601.439,Z 204.562,A -85,B 0,C 180,E1 -711.939,E2 -711.939} C_VEL
LIN {X 0,Y 601.43,Z 204.573,A -85,B 0,C 180,E1 -714.636,E2 -714.636} C_VEL
LIN {X 0,Y 601.419,Z 204.564,A -85,B 0,C 180,E1 -717.321,E2 -717.321} C_VEL
LIN {X 0,Y 601.445,Z 204.562,A -85,B 0,C 180,E1 -720,E2 -720} C_VEL
LIN {X 0,Y 601.445,Z 204.57,A -85,B 0,C 180,E1 -722.679,E2 -722.679} C_VEL
LIN {X 0,Y 601.406,Z 204.565,A -85,B 0,C 180,E1 -725.364,E2 -725.364} C_VEL
LIN {X 0,Y 601.44,Z 204.563,A -85,B 0,C 180,E1 -728.061,E2 -728.061} C_VEL
LIN {X 0,Y 601.423,Z 204.567,A -85,B 0,C 180,E1 -731.011,E2 -731.011} C_VEL
LIN {X 0,Y 601.403,Z 204.565,A -85,B 0,C 180,E1 -733.516,E2 -733.516} C_VEL
LIN {X 0,Y 601.44,Z 204.566,A -85,B 0,C 180,E1 -736.287,E2 -736.287} C_VEL
LIN {X 0,Y 601.411,Z 204.567,A -85,B 0,C 180,E1 -739.099,E2 -739.099} C_VEL
LIN {X 0,Y 601.397,Z 204.567,A -85,B 0,C 180,E1 -741.24,E2 -741.24} C_VEL
LIN {X 0,Y 601.462,Z 204.561,A -85,B 0,C 180,E1 -744.14,E2 -744.14} C_VEL
LIN {X 0,Y 601.396,Z 204.568,A -85,B 0,C 180,E1 -747.114,E2 -747.114} C_VEL
LIN {X 0,Y 601.397,Z 204.566,A -85,B 0,C 180,E1 -749.394,E2 -749.394} C_VEL
LIN {X 0,Y 601.398,Z 204.566,A -85,B 0,C 180,E1 -751.727,E2 -751.727} C_VEL
LIN {X 0,Y 601.421,Z 204.566,A -85,B 0,C 180,E1 -754.119,E2 -754.119} C_VEL
LIN {X 0,Y 601.392,Z 204.577,A -85,B 0,C 180,E1 -756.584,E2 -756.584} C_VEL
LIN {X 0,Y 601.396,Z 204.568,A -85,B 0,C 180,E1 -759.128,E2 -759.128} C_VEL
LIN {X 0,Y 601.42,Z 204.564,A -85,B 0,C 180,E1 -761.766,E2 -761.766} C_VEL
LIN {X 0,Y 601.398,Z 204.577,A -85,B 0,C 180,E1 -764.533,E2 -764.533} C_VEL
LIN {X 0,Y 601.43,Z 204.571,A -85,B 0,C 180,E1 -766.427,E2 -766.427} C_VEL
LIN {X 0,Y 601.404,Z 204.567,A -85,B 0,C 180,E1 -769.125,E2 -769.125} C_VEL
LIN {X 0,Y 601.41,Z 204.565,A -85,B 0,C 180,E1 -771.731,E2 -771.731} C_VEL
LIN {X 0,Y 601.387,Z 204.573,A -85,B 0,C 180,E1 -774.245,E2 -774.245} C_VEL
LIN {X 0,Y 601.425,Z 204.571,A -85,B 0,C 180,E1 -776.686,E2 -776.686} C_VEL
LIN {X 0,Y 601.398,Z 204.568,A -85,B 0,C 180,E1 -779.057,E2 -779.057} C_VEL
LIN {X 0,Y 601.406,Z 204.565,A -85,B 0,C 180,E1 -781.372,E2 -781.372} C_VEL
LIN {X 0,Y 601.41,Z 204.569,A -85,B 0,C 180,E1 -784.134,E2 -784.134} C_VEL
LIN {X 0,Y 601.392,Z 204.577,A -85,B 0,C 180,E1 -786.589,E2 -786.589} C_VEL
LIN {X 0,Y 601.403,Z 204.617,A -85,B 0,C 180,E1 -787.557,E2 -787.557} C_VEL
LIN {X 0,Y 601.636,Z 211.761,A -85,B 0,C 180,E1 -788.59,E2 -788.59} C_VEL
LIN {X 0,Y 601.535,Z 231.492,A -85,B 0,C 180,E1 -791.377,E2 -791.377} C_VEL
LIN {X 0,Y 601.483,Z 250.801,A -85,B 0,C 180,E1 -794.063,E2 -794.063} C_VEL
LIN {X 0,Y 601.445,Z 270.792,A -85,B 0,C 180,E1 -796.807,E2 -796.807} C_VEL
LIN {X 0,Y 601.651,Z 276.51,A -85,B 0,C 180,E1 -796.898,E2 -796.898} C_VEL
LIN {X 0,Y 601.602,Z 378.948,A -85,B 0,C 180,E1 -798.139,E2 -798.139} C_VEL
LIN {X 0,Y 601.562,Z 392.218,A -85,B 0,C 180,E1 -798.438,E2 -798.438} C_VEL
LIN {X 0,Y 601.536,Z 403.953,A -85,B 0,C 180,E1 -798.827,E2 -798.827} C_VEL
LIN {X 0,Y 601.526,Z 414.924,A -85,B 0,C 180,E1 -799.311,E2 -799.311} C_VEL
LIN {X 0,Y 601.484,Z 425.581,A -85,B 0,C 180,E1 -799.906,E2 -799.906} C_VEL
LIN {X 0,Y 601.448,Z 436.476,A -85,B 0,C 180,E1 -800.669,E2 -800.669} C_VEL
LIN {X 0,Y 601.429,Z 447.112,A -85,B 0,C 180,E1 -801.601,E2 -801.601} C_VEL
LIN {X 0,Y 601.418,Z 454.961,A -85,B 0,C 180,E1 -802.446,E2 -802.446} C_VEL
LIN {X 0,Y 601.37,Z 462.225,A -85,B 0,C 180,E1 -803.398,E2 -803.398} C_VEL
LIN {X 0,Y 601.372,Z 467.866,A -85,B 0,C 180,E1 -804.299,E2 -804.299} C_VEL
LIN {X 0,Y 601.336,Z 472.95,A -85,B 0,C 180,E1 -805.307,E2 -805.307} C_VEL
LIN {X 0,Y 601.368,Z 476.896,A -85,B 0,C 180,E1 -806.315,E2 -806.315} C_VEL
LIN {X 0,Y 601.325,Z 479.809,A -85,B 0,C 180,E1 -807.32,E2 -807.32} C_VEL
LIN {X 0,Y 601.343,Z 481.202,A -85,B 0,C 180,E1 -807.991,E2 -807.991} C_VEL
LIN {X 0,Y 601.339,Z 482.784,A -85,B 0,C 180,E1 -809.33,E2 -809.33} C_VEL
LIN {X 0,Y 601.335,Z 483,A -85,B 0,C 180,E1 -810,E2 -810} C_VEL
LIN {X 0,Y 601.347,Z 482.184,A -85,B 0,C 180,E1 -811.339,E2 -811.339} C_VEL
LIN {X 0,Y 601.343,Z 481.202,A -85,B 0,C 180,E1 -812.009,E2 -812.009} C_VEL
LIN {X 0,Y 601.325,Z 479.809,A -85,B 0,C 180,E1 -812.68,E2 -812.68} C_VEL
LIN {X 0,Y 601.368,Z 476.896,A -85,B 0,C 180,E1 -813.685,E2 -813.685} C_VEL
LIN {X 0,Y 601.336,Z 472.95,A -85,B 0,C 180,E1 -814.693,E2 -814.693} C_VEL
LIN {X 0,Y 601.372,Z 466.877,A -85,B 0,C 180,E1 -815.869,E2 -815.869} C_VEL
LIN {X 0,Y 601.382,Z 460.235,A -85,B 0,C 180,E1 -816.88,E2 -816.88} C_VEL
LIN {X 0,Y 601.401,Z 451.989,A -85,B 0,C 180,E1 -817.892,E2 -817.892} C_VEL
LIN {X 0,Y 601.436,Z 443.536,A -85,B 0,C 180,E1 -818.738,E2 -818.738} C_VEL
LIN {X 0,Y 601.448,Z 433.092,A -85,B 0,C 180,E1 -819.585,E2 -819.585} C_VEL
LIN {X 0,Y 601.478,Z 422.757,A -85,B 0,C 180,E1 -820.264,E2 -820.264} C_VEL
LIN {X 0,Y 601.535,Z 411.91,A -85,B 0,C 180,E1 -820.835,E2 -820.835} C_VEL
LIN {X 0,Y 601.544,Z 399.382,A -85,B 0,C 180,E1 -821.341,E2 -821.341} C_VEL
LIN {X 0,Y 601.554,Z 386.35,A -85,B 0,C 180,E1 -821.712,E2 -821.712} C_VEL
LIN {X 0,Y 601.61,Z 373.082,A -85,B 0,C 180,E1 -821.946,E2 -821.946} C_VEL
LIN {X 0,Y 601.551,Z 271.81,A -85,B 0,C 180,E1 -823.161,E2 -823.161} C_VEL
LIN {X 0,Y 601.457,Z 270.635,A -85,B 0,C 180,E1 -823.214,E2 -823.214} C_VEL
LIN {X 0,Y 601.484,Z 250.8,A -85,B 0,C 180,E1 -825.937,E2 -825.937} C_VEL
LIN {X 0,Y 601.535,Z 231.495,A -85,B 0,C 180,E1 -828.623,E2 -828.623} C_VEL
LIN {X 0,Y 601.636,Z 211.761,A -85,B 0,C 180,E1 -831.41,E2 -831.41} C_VEL
LIN {X 0,Y 601.403,Z 204.617,A -85,B 0,C 180,E1 -832.443,E2 -832.443} C_VEL
LIN {X 0,Y 601.39,Z 204.569,A -85,B 0,C 180,E1 -834.879,E2 -834.879} C_VEL
LIN {X 0,Y 601.395,Z 204.571,A -85,B 0,C 180,E1 -837.869,E2 -837.869} C_VEL
LIN {X 0,Y 601.407,Z 204.566,A -85,B 0,C 180,E1 -840.165,E2 -840.165} C_VEL
LIN {X 0,Y 601.404,Z 204.566,A -85,B 0,C 180,E1 -842.712,E2 -842.712} C_VEL
LIN {X 0,Y 601.381,Z 204.573,A -85,B 0,C 180,E1 -845.11,E2 -845.11} C_VEL
LIN {X 0,Y 601.432,Z 204.572,A -85,B 0,C 180,E1 -847.419,E2 -847.419} C_VEL
LIN {X 0,Y 601.402,Z 204.568,A -85,B 0,C 180,E1 -849.996,E2 -849.996} C_VEL
LIN {X 0,Y 601.377,Z 204.569,A -85,B 0,C 180,E1 -852.673,E2 -852.673} C_VEL
LIN {X 0,Y 601.399,Z 204.566,A -85,B 0,C 180,E1 -854.532,E2 -854.532} C_VEL
LIN {X 0,Y 601.411,Z 204.575,A -85,B 0,C 180,E1 -857.409,E2 -857.409} C_VEL
LIN {X 0,Y 601.401,Z 204.568,A -85,B 0,C 180,E1 -860.004,E2 -860.004} C_VEL
LIN {X 0,Y 601.4,Z 204.566,A -85,B 0,C 180,E1 -862.622,E2 -862.622} C_VEL
LIN {X 0,Y 601.397,Z 204.57,A -85,B 0,C 180,E1 -865.067,E2 -865.067} C_VEL
LIN {X 0,Y 601.434,Z 204.572,A -85,B 0,C 180,E1 -867.484,E2 -867.484} C_VEL
LIN {X 0,Y 601.429,Z 204.566,A -85,B 0,C 180,E1 -869.852,E2 -869.852} C_VEL
LIN {X 0,Y 601.386,Z 204.568,A -85,B 0,C 180,E1 -872.643,E2 -872.643} C_VEL
LIN {X 0,Y 601.389,Z 204.572,A -85,B 0,C 180,E1 -875.121,E2 -875.121} C_VEL
LIN {X 0,Y 601.416,Z 204.574,A -85,B 0,C 180,E1 -877.395,E2 -877.395} C_VEL
LIN {X 0,Y 601.396,Z 204.567,A -85,B 0,C 180,E1 -880.19,E2 -880.19} C_VEL
LIN {X 0,Y 601.386,Z 204.567,A -85,B 0,C 180,E1 -882.311,E2 -882.311} C_VEL
LIN {X 0,Y 601.397,Z 204.566,A -85,B 0,C 180,E1 -884.408,E2 -884.408} C_VEL
LIN {X 0,Y 601.412,Z 204.57,A -85,B 0,C 180,E1 -887.172,E2 -887.172} C_VEL
LIN {X 0,Y 601.431,Z 204.565,A -85,B 0,C 180,E1 -889.905,E2 -889.905} C_VEL
LIN {X 0,Y 601.398,Z 204.566,A -85,B 0,C 180,E1 -892.614,E2 -892.614} C_VEL
LIN {X 0,Y 601.426,Z 204.571,A -85,B 0,C 180,E1 -895.308,E2 -895.308} C_VEL
LIN {X 0,Y 601.435,Z 204.563,A -85,B 0,C 180,E1 -897.991,E2 -897.991} C_VEL
LIN {X 0,Y 601.426,Z 204.563,A -85,B 0,C 180,E1 -900.67,E2 -900.67} C_VEL
LIN {X 0,Y 601.424,Z 204.572,A -85,B 0,C 180,E1 -903.35,E2 -903.35} C_VEL
LIN {X 0,Y 601.432,Z 204.563,A -85,B 0,C 180,E1 -906.037,E2 -906.037} C_VEL
LIN {X 0,Y 601.397,Z 204.567,A -85,B 0,C 180,E1 -908.738,E2 -908.738} C_VEL
LIN {X 0,Y 601.423,Z 204.573,A -85,B 0,C 180,E1 -911.458,E2 -911.458} C_VEL
LIN {X 0,Y 601.4,Z 204.565,A -85,B 0,C 180,E1 -912.348,E2 -912.348} C_VEL
LIN {X 0,Y 600.724,Z 204.654,A -85,B 0,C 180,E1 -912.907,E2 -912.907} C_VEL
LIN {X 0,Y 597.867,Z 205.01,A -85,B 0,C 180,E1 -913.815,E2 -913.815} C_VEL
LIN {X 0,Y 595.46,Z 205.31,A -85,B 0,C 180,E1 -914.546,E2 -914.546} C_VEL
LIN {X 0,Y 594.428,Z 205.439,A -85,B 0,C 180,E1 -915.109,E2 -915.109} C_VEL
LIN {X 0,Y 594.345,Z 205.448,A -85,B 0,C 180,E1 -915.3,E2 -915.3} C_VEL
LIN {X 0,Y 594.343,Z 205.447,A -85,B 0,C 180,E1 -917.905,E2 -917.905} C_VEL
LIN {X 0,Y 594.386,Z 205.441,A -85,B 0,C 180,E1 -920.776,E2 -920.776} C_VEL
LIN {X 0,Y 594.379,Z 205.446,A -85,B 0,C 180,E1 -923.705,E2 -923.705} C_VEL
LIN {X 0,Y 594.361,Z 205.444,A -85,B 0,C 180,E1 -926.018,E2 -926.018} C_VEL
LIN {X 0,Y 594.363,Z 205.443,A -85,B 0,C 180,E1 -928.228,E2 -928.228} C_VEL
LIN {X 0,Y 594.368,Z 205.442,A -85,B 0,C 180,E1 -930.561,E2 -930.561} C_VEL
LIN {X 0,Y 594.377,Z 205.444,A -85,B 0,C 180,E1 -932.951,E2 -932.951} C_VEL
LIN {X 0,Y 594.348,Z 205.455,A -85,B 0,C 180,E1 -935.409,E2 -935.409} C_VEL
LIN {X 0,Y 594.382,Z 205.442,A -85,B 0,C 180,E1 -937.941,E2 -937.941} C_VEL
LIN {X 0,Y 594.37,Z 205.443,A -85,B 0,C 180,E1 -940.821,E2 -940.821} C_VEL
LIN {X 0,Y 594.363,Z 205.446,A -85,B 0,C 180,E1 -943.839,E2 -943.839} C_VEL
LIN {X 0,Y 594.352,Z 205.444,A -85,B 0,C 180,E1 -946.699,E2 -946.699} C_VEL
LIN {X 0,Y 594.37,Z 205.452,A -85,B 0,C 180,E1 -949.433,E2 -949.433} C_VEL
LIN {X 0,Y 594.388,Z 205.44,A -85,B 0,C 180,E1 -952.392,E2 -952.392} C_VEL
LIN {X 0,Y 594.374,Z 205.452,A -85,B 0,C 180,E1 -955.42,E2 -955.42} C_VEL
LIN {X 0,Y 594.375,Z 205.441,A -85,B 0,C 180,E1 -958.358,E2 -958.358} C_VEL
LIN {X 0,Y 594.382,Z 205.445,A -85,B 0,C 180,E1 -961.043,E2 -961.043} C_VEL
LIN {X 0,Y 594.364,Z 205.445,A -85,B 0,C 180,E1 -964.055,E2 -964.055} C_VEL
LIN {X 0,Y 594.37,Z 205.526,A -85,B 0,C 180,E1 -964.549,E2 -964.549} C_VEL
LIN {X 0,Y 594.465,Z 215.775,A -85,B 0,C 180,E1 -966.299,E2 -966.299} C_VEL
LIN {X 0,Y 594.415,Z 230.817,A -85,B 0,C 180,E1 -968.832,E2 -968.832} C_VEL
LIN {X 0,Y 594.341,Z 242.143,A -85,B 0,C 180,E1 -970.718,E2 -970.718} C_VEL
LIN {X 0,Y 594.742,Z 246.183,A -85,B 0,C 180,E1 -970.784,E2 -970.784} C_VEL
LIN {X 0,Y 594.638,Z 348.601,A -85,B 0,C 180,E1 -972.037,E2 -972.037} C_VEL
LIN {X 0,Y 594.603,Z 361.497,A -85,B 0,C 180,E1 -972.325,E2 -972.325} C_VEL
LIN {X 0,Y 594.577,Z 374.69,A -85,B 0,C 180,E1 -972.768,E2 -972.768} C_VEL
LIN {X 0,Y 594.539,Z 385.736,A -85,B 0,C 180,E1 -973.269,E2 -973.269} C_VEL
LIN {X 0,Y 594.47,Z 397.534,A -85,B 0,C 180,E1 -973.958,E2 -973.958} C_VEL
LIN {X 0,Y 594.4,Z 408.262,A -85,B 0,C 180,E1 -974.747,E2 -974.747} C_VEL
LIN {X 0,Y 594.377,Z 417.892,A -85,B 0,C 180,E1 -975.623,E2 -975.623} C_VEL
LIN {X 0,Y 594.315,Z 427.105,A -85,B 0,C 180,E1 -976.668,E2 -976.668} C_VEL
LIN {X 0,Y 594.29,Z 434.494,A -85,B 0,C 180,E1 -977.71,E2 -977.71} C_VEL
LIN {X 0,Y 594.311,Z 440.373,A -85,B 0,C 180,E1 -978.749,E2 -978.749} C_VEL
LIN {X 0,Y 594.25,Z 444.966,A -85,B 0,C 180,E1 -979.782,E2 -979.782} C_VEL
LIN {X 0,Y 594.266,Z 447.38,A -85,B 0,C 180,E1 -980.47,E2 -980.47} C_VEL
LIN {X 0,Y 594.231,Z 449.348,A -85,B 0,C 180,E1 -981.156,E2 -981.156} C_VEL
LIN {X 0,Y 594.23,Z 450.896,A -85,B 0,C 180,E1 -981.841,E2 -981.841} C_VEL
LIN {X 0,Y 594.247,Z 451.994,A -85,B 0,C 180,E1 -982.525,E2 -982.525} C_VEL
LIN {X 0,Y 594.263,Z 452.824,A -85,B 0,C 180,E1 -983.426,E2 -983.426} C_VEL
LIN {X 0,Y 594.25,Z 452.88,A -85,B 0,C 180,E1 -984.571,E2 -984.571} C_VEL
LIN {X 0,Y 594.255,Z 451.441,A -85,B 0,C 180,E1 -985.931,E2 -985.931} C_VEL
LIN {X 0,Y 594.259,Z 450.133,A -85,B 0,C 180,E1 -986.61,E2 -986.61} C_VEL
LIN {X 0,Y 594.255,Z 447.356,A -85,B 0,C 180,E1 -987.628,E2 -987.628} C_VEL
LIN {X 0,Y 594.256,Z 443.574,A -85,B 0,C 180,E1 -988.645,E2 -988.645} C_VEL
LIN {X 0,Y 594.299,Z 438.681,A -85,B 0,C 180,E1 -989.661,E2 -989.661} C_VEL
LIN {X 0,Y 594.295,Z 432.543,A -85,B 0,C 180,E1 -990.678,E2 -990.678} C_VEL
LIN {X 0,Y 594.355,Z 424.923,A -85,B 0,C 180,E1 -991.694,E2 -991.694} C_VEL
LIN {X 0,Y 594.366,Z 415.389,A -85,B 0,C 180,E1 -992.711,E2 -992.711} C_VEL
LIN {X 0,Y 594.432,Z 405.579,A -85,B 0,C 180,E1 -993.559,E2 -993.559} C_VEL
LIN {X 0,Y 594.482,Z 394.551,A -85,B 0,C 180,E1 -994.322,E2 -994.322} C_VEL
LIN {X 0,Y 594.55,Z 383.803,A -85,B 0,C 180,E1 -994.916,E2 -994.916} C_VEL
LIN {X 0,Y 594.558,Z 371.994,A -85,B 0,C 180,E1 -995.426,E2 -995.426} C_VEL
LIN {X 0,Y 594.628,Z 359.135,A -85,B 0,C 180,E1 -995.83,E2 -995.83} C_VEL
LIN {X 0,Y 594.667,Z 346.441,A -85,B 0,C 180,E1 -996.085,E2 -996.085} C_VEL
LIN {X 0,Y 594.652,Z 244.078,A -85,B 0,C 180,E1 -997.334,E2 -997.334} C_VEL
LIN {X 0,Y 594.37,Z 242.045,A -85,B 0,C 180,E1 -997.388,E2 -997.388} C_VEL
LIN {X 0,Y 594.458,Z 226.134,A -85,B 0,C 180,E1 -1000.043,E2 -1000.043} C_VEL
LIN {X 0,Y 594.542,Z 208.777,A -85,B 0,C 180,E1 -1002.979,E2 -1002.979} C_VEL
LIN {X 0,Y 594.363,Z 205.446,A -85,B 0,C 180,E1 -1003.592,E2 -1003.592} C_VEL
LIN {X 0,Y 594.413,Z 205.444,A -85,B 0,C 180,E1 -1006.485,E2 -1006.485} C_VEL
LIN {X 0,Y 594.366,Z 205.443,A -85,B 0,C 180,E1 -1009.334,E2 -1009.334} C_VEL
LIN {X 0,Y 594.363,Z 205.443,A -85,B 0,C 180,E1 -1011.503,E2 -1011.503} C_VEL
LIN {X 0,Y 594.393,Z 205.445,A -85,B 0,C 180,E1 -1014.446,E2 -1014.446} C_VEL
LIN {X 0,Y 594.362,Z 205.453,A -85,B 0,C 180,E1 -1016.701,E2 -1016.701} C_VEL
LIN {X 0,Y 594.379,Z 205.445,A -85,B 0,C 180,E1 -1018.999,E2 -1018.999} C_VEL
LIN {X 0,Y 594.376,Z 205.441,A -85,B 0,C 180,E1 -1021.642,E2 -1021.642} C_VEL
LIN {X 0,Y 594.379,Z 205.449,A -85,B 0,C 180,E1 -1024.58,E2 -1024.58} C_VEL
LIN {X 0,Y 594.389,Z 205.439,A -85,B 0,C 180,E1 -1027.608,E2 -1027.608} C_VEL
LIN {X 0,Y 594.37,Z 205.45,A -85,B 0,C 180,E1 -1030.567,E2 -1030.567} C_VEL
LIN {X 0,Y 594.353,Z 205.445,A -85,B 0,C 180,E1 -1033.301,E2 -1033.301} C_VEL
LIN {X 0,Y 594.363,Z 205.445,A -85,B 0,C 180,E1 -1036.161,E2 -1036.161} C_VEL
LIN {X 0,Y 594.373,Z 205.444,A -85,B 0,C 180,E1 -1039.179,E2 -1039.179} C_VEL
LIN {X 0,Y 594.382,Z 205.442,A -85,B 0,C 180,E1 -1042.059,E2 -1042.059} C_VEL
LIN {X 0,Y 594.349,Z 205.455,A -85,B 0,C 180,E1 -1044.677,E2 -1044.677} C_VEL
LIN {X 0,Y 594.377,Z 205.444,A -85,B 0,C 180,E1 -1047.089,E2 -1047.089} C_VEL
LIN {X 0,Y 594.387,Z 205.439,A -85,B 0,C 180,E1 -1049.672,E2 -1049.672} C_VEL
LIN {X 0,Y 594.376,Z 205.45,A -85,B 0,C 180,E1 -1052.539,E2 -1052.539} C_VEL
LIN {X 0,Y 594.372,Z 205.449,A -85,B 0,C 180,E1 -1054.807,E2 -1054.807} C_VEL
LIN {X 0,Y 594.36,Z 205.444,A -85,B 0,C 180,E1 -1057.266,E2 -1057.266} C_VEL
LIN {X 0,Y 594.368,Z 205.443,A -85,B 0,C 180,E1 -1059.946,E2 -1059.946} C_VEL
LIN {X 0,Y 594.378,Z 205.448,A -85,B 0,C 180,E1 -1062.806,E2 -1062.806} C_VEL
LIN {X 0,Y 594.388,Z 205.439,A -85,B 0,C 180,E1 -1065.827,E2 -1065.827} C_VEL
LIN {X 0,Y 594.394,Z 205.445,A -85,B 0,C 180,E1 -1068.404,E2 -1068.404} C_VEL
LIN {X 0,Y 594.369,Z 205.444,A -85,B 0,C 180,E1 -1071.158,E2 -1071.158} C_VEL
LIN {X 0,Y 594.379,Z 205.441,A -85,B 0,C 180,E1 -1073.891,E2 -1073.891} C_VEL
LIN {X 0,Y 594.379,Z 205.451,A -85,B 0,C 180,E1 -1076.611,E2 -1076.611} C_VEL
LIN {X 0,Y 594.401,Z 205.438,A -85,B 0,C 180,E1 -1079.322,E2 -1079.322} C_VEL
LIN {X 0,Y 594.404,Z 205.439,A -85,B 0,C 180,E1 -1082.033,E2 -1082.033} C_VEL
LIN {X 0,Y 594.393,Z 205.447,A -85,B 0,C 180,E1 -1084.748,E2 -1084.748} C_VEL
LIN {X 0,Y 594.366,Z 205.442,A -85,B 0,C 180,E1 -1087.473,E2 -1087.473} C_VEL
LIN {X 0,Y 594.391,Z 205.443,A -85,B 0,C 180,E1 -1090.216,E2 -1090.216} C_VEL
LIN {X 0,Y 594.36,Z 205.447,A -85,B 0,C 180,E1 -1092.983,E2 -1092.983} C_VEL
LIN {X 0,Y 594.364,Z 205.445,A -85,B 0,C 180,E1 -1095.078,E2 -1095.078} C_VEL
LIN {X 0,Y 594.375,Z 205.442,A -85,B 0,C 180,E1 -1097.194,E2 -1097.194} C_VEL
LIN {X 0,Y 594.37,Z 205.444,A -85,B 0,C 180,E1 -1100.054,E2 -1100.054} C_VEL
LIN {X 0,Y 594.355,Z 205.447,A -85,B 0,C 180,E1 -1102.968,E2 -1102.968} C_VEL
LIN {X 0,Y 594.356,Z 205.445,A -85,B 0,C 180,E1 -1105.194,E2 -1105.194} C_VEL
LIN {X 0,Y 594.342,Z 205.445,A -85,B 0,C 180,E1 -1107.518,E2 -1107.518} C_VEL
LIN {X 0,Y 594.386,Z 205.446,A -85,B 0,C 180,E1 -1110.328,E2 -1110.328} C_VEL
LIN {X 0,Y 594.376,Z 205.445,A -85,B 0,C 180,E1 -1112.95,E2 -1112.95} C_VEL
LIN {X 0,Y 594.346,Z 205.445,A -85,B 0,C 180,E1 -1115.409,E2 -1115.409} C_VEL
LIN {X 0,Y 594.384,Z 205.441,A -85,B 0,C 180,E1 -1117.941,E2 -1117.941} C_VEL
LIN {X 0,Y 594.367,Z 205.448,A -85,B 0,C 180,E1 -1120.821,E2 -1120.821} C_VEL
LIN {X 0,Y 594.35,Z 205.444,A -85,B 0,C 180,E1 -1123.301,E2 -1123.301} C_VEL
LIN {X 0,Y 594.361,Z 205.447,A -85,B 0,C 180,E1 -1126.161,E2 -1126.161} C_VEL
LIN {X 0,Y 594.38,Z 205.451,A -85,B 0,C 180,E1 -1128.536,E2 -1128.536} C_VEL
LIN {X 0,Y 594.368,Z 205.442,A -85,B 0,C 180,E1 -1131.298,E2 -1131.298} C_VEL
LIN {X 0,Y 594.348,Z 205.445,A -85,B 0,C 180,E1 -1133.755,E2 -1133.755} C_VEL
LIN {X 0,Y 594.38,Z 205.446,A -85,B 0,C 180,E1 -1136.239,E2 -1136.239} C_VEL
LIN {X 0,Y 594.365,Z 205.451,A -85,B 0,C 180,E1 -1138.649,E2 -1138.649} C_VEL
LIN {X 0,Y 594.376,Z 205.444,A -85,B 0,C 180,E1 -1141.044,E2 -1141.044} C_VEL
LIN {X 0,Y 594.363,Z 205.443,A -85,B 0,C 180,E1 -1143.299,E2 -1143.299} C_VEL
LIN {X 0,Y 594.359,Z 205.443,A -85,B 0,C 180,E1 -1145.573,E2 -1145.573} C_VEL
LIN {X 0,Y 594.379,Z 205.551,A -85,B 0,C 180,E1 -1147.413,E2 -1147.413} C_VEL
LIN {X 0,Y 594.745,Z 209.243,A -85,B 0,C 180,E1 -1147.964,E2 -1147.964} C_VEL
LIN {X 0,Y 594.628,Z 229.72,A -85,B 0,C 180,E1 -1150.9,E2 -1150.9} C_VEL
LIN {X 0,Y 594.5,Z 249.541,A -85,B 0,C 180,E1 -1153.694,E2 -1153.694} C_VEL
LIN {X 0,Y 594.423,Z 269.691,A -85,B 0,C 180,E1 -1156.496,E2 -1156.496} C_VEL
LIN {X 0,Y 594.46,Z 271.144,A -85,B 0,C 180,E1 -1156.671,E2 -1156.671} C_VEL
LIN {X 0,Y 594.74,Z 280.087,A -85,B 0,C 180,E1 -1156.786,E2 -1156.786} C_VEL
LIN {X 0,Y 594.654,Z 378.948,A -85,B 0,C 180,E1 -1157.999,E2 -1157.999} C_VEL
LIN {X 0,Y 594.626,Z 392.219,A -85,B 0,C 180,E1 -1158.301,E2 -1158.301} C_VEL
LIN {X 0,Y 594.57,Z 404.571,A -85,B 0,C 180,E1 -1158.718,E2 -1158.718} C_VEL
LIN {X 0,Y 594.533,Z 416.632,A -85,B 0,C 180,E1 -1159.27,E2 -1159.27} C_VEL
LIN {X 0,Y 594.472,Z 428.201,A -85,B 0,C 180,E1 -1159.958,E2 -1159.958} C_VEL
LIN {X 0,Y 594.414,Z 438.597,A -85,B 0,C 180,E1 -1160.73,E2 -1160.73} C_VEL
LIN {X 0,Y 594.383,Z 447.112,A -85,B 0,C 180,E1 -1161.501,E2 -1161.501} C_VEL
LIN {X 0,Y 594.347,Z 454.961,A -85,B 0,C 180,E1 -1162.355,E2 -1162.355} C_VEL
LIN {X 0,Y 594.283,Z 462.813,A -85,B 0,C 180,E1 -1163.408,E2 -1163.408} C_VEL
LIN {X 0,Y 594.289,Z 469.68,A -85,B 0,C 180,E1 -1164.571,E2 -1164.571} C_VEL
LIN {X 0,Y 594.27,Z 474.371,A -85,B 0,C 180,E1 -1165.591,E2 -1165.591} C_VEL
LIN {X 0,Y 594.267,Z 477.956,A -85,B 0,C 180,E1 -1166.61,E2 -1166.61} C_VEL
LIN {X 0,Y 594.226,Z 479.809,A -85,B 0,C 180,E1 -1167.288,E2 -1167.288} C_VEL
LIN {X 0,Y 594.241,Z 481.201,A -85,B 0,C 180,E1 -1167.967,E2 -1167.967} C_VEL
LIN {X 0,Y 594.239,Z 482.784,A -85,B 0,C 180,E1 -1169.322,E2 -1169.322} C_VEL
LIN {X 0,Y 594.236,Z 483,A -85,B 0,C 180,E1 -1170,E2 -1170} C_VEL
LIN {X 0,Y 594.247,Z 482.185,A -85,B 0,C 180,E1 -1171.355,E2 -1171.355} C_VEL
LIN {X 0,Y 594.241,Z 481.201,A -85,B 0,C 180,E1 -1172.033,E2 -1172.033} C_VEL
LIN {X 0,Y 594.226,Z 479.81,A -85,B 0,C 180,E1 -1172.712,E2 -1172.712} C_VEL
LIN {X 0,Y 594.289,Z 476.896,A -85,B 0,C 180,E1 -1173.729,E2 -1173.729} C_VEL
LIN {X 0,Y 594.241,Z 472.949,A -85,B 0,C 180,E1 -1174.749,E2 -1174.749} C_VEL
LIN {X 0,Y 594.304,Z 466.877,A -85,B 0,C 180,E1 -1175.939,E2 -1175.939} C_VEL
LIN {X 0,Y 594.308,Z 460.236,A -85,B 0,C 180,E1 -1176.962,E2 -1176.962} C_VEL
LIN {X 0,Y 594.359,Z 451.99,A -85,B 0,C 180,E1 -1177.986,E2 -1177.986} C_VEL
LIN {X 0,Y 594.382,Z 443.537,A -85,B 0,C 180,E1 -1178.842,E2 -1178.842} C_VEL
LIN {X 0,Y 594.431,Z 433.094,A -85,B 0,C 180,E1 -1179.699,E2 -1179.699} C_VEL
LIN {X 0,Y 594.489,Z 422.758,A -85,B 0,C 180,E1 -1180.386,E2 -1180.386} C_VEL
LIN {X 0,Y 594.559,Z 411.71,A -85,B 0,C 180,E1 -1180.974,E2 -1180.974} C_VEL
LIN {X 0,Y 594.573,Z 399.706,A -85,B 0,C 180,E1 -1181.464,E2 -1181.464} C_VEL
LIN {X 0,Y 594.607,Z 386.349,A -85,B 0,C 180,E1 -1181.851,E2 -1181.851} C_VEL
LIN {X 0,Y 594.662,Z 373.082,A -85,B 0,C 180,E1 -1182.088,E2 -1182.088} C_VEL
LIN {X 0,Y 594.702,Z 272.928,A -85,B 0,C 180,E1 -1183.302,E2 -1183.302} C_VEL
LIN {X 0,Y 594.422,Z 270.792,A -85,B 0,C 180,E1 -1183.351,E2 -1183.351} C_VEL
LIN {X 0,Y 594.502,Z 250.8,A -85,B 0,C 180,E1 -1186.129,E2 -1186.129} C_VEL
LIN {X 0,Y 594.598,Z 231.308,A -85,B 0,C 180,E1 -1188.875,E2 -1188.875} C_VEL
LIN {X 0,Y 594.751,Z 211.761,A -85,B 0,C 180,E1 -1191.671,E2 -1191.671} C_VEL
LIN {X 0,Y 594.463,Z 206.028,A -85,B 0,C 180,E1 -1192.514,E2 -1192.514} C_VEL
LIN {X 0,Y 594.378,Z 205.446,A -85,B 0,C 180,E1 -1192.621,E2 -1192.621} C_VEL
LIN {X 0,Y 594.371,Z 205.448,A -85,B 0,C 180,E1 -1195.193,E2 -1195.193} C_VEL
LIN {X 0,Y 594.37,Z 205.452,A -85,B 0,C 180,E1 -1197.523,E2 -1197.523} C_VEL
LIN {X 0,Y 594.371,Z 205.442,A -85,B 0,C 180,E1 -1200.325,E2 -1200.325} C_VEL
LIN {X 0,Y 594.376,Z 205.443,A -85,B 0,C 180,E1 -1202.95,E2 -1202.95} C_VEL
LIN {X 0,Y 594.347,Z 205.454,A -85,B 0,C 180,E1 -1205.409,E2 -1205.409} C_VEL
LIN {X 0,Y 594.381,Z 205.443,A -85,B 0,C 180,E1 -1207.941,E2 -1207.941} C_VEL
LIN {X 0,Y 594.367,Z 205.443,A -85,B 0,C 180,E1 -1210.821,E2 -1210.821} C_VEL
LIN {X 0,Y 594.359,Z 205.451,A -85,B 0,C 180,E1 -1213.3,E2 -1213.3} C_VEL
LIN {X 0,Y 594.344,Z 205.446,A -85,B 0,C 180,E1 -1216.163,E2 -1216.163} C_VEL
LIN {X 0,Y 594.369,Z 205.442,A -85,B 0,C 180,E1 -1218.535,E2 -1218.535} C_VEL
LIN {X 0,Y 594.378,Z 205.448,A -85,B 0,C 180,E1 -1221.297,E2 -1221.297} C_VEL
LIN {X 0,Y 594.35,Z 205.449,A -85,B 0,C 180,E1 -1223.755,E2 -1223.755} C_VEL
LIN {X 0,Y 594.364,Z 205.442,A -85,B 0,C 180,E1 -1226.238,E2 -1226.238} C_VEL
LIN {X 0,Y 594.364,Z 205.443,A -85,B 0,C 180,E1 -1228.649,E2 -1228.649} C_VEL
LIN {X 0,Y 594.379,Z 205.444,A -85,B 0,C 180,E1 -1231.043,E2 -1231.043} C_VEL
LIN {X 0,Y 594.363,Z 205.444,A -85,B 0,C 180,E1 -1234.055,E2 -1234.055} C_VEL
LIN {X 0,Y 594.375,Z 205.441,A -85,B 0,C 180,E1 -1236.295,E2 -1236.295} C_VEL
LIN {X 0,Y 594.403,Z 205.444,A -85,B 0,C 180,E1 -1239.224,E2 -1239.224} C_VEL
LIN {X 0,Y 594.349,Z 205.445,A -85,B 0,C 180,E1 -1242.095,E2 -1242.095} C_VEL
LIN {X 0,Y 594.355,Z 205.444,A -85,B 0,C 180,E1 -1244.219,E2 -1244.219} C_VEL
LIN {X 0,Y 594.372,Z 205.441,A -85,B 0,C 180,E1 -1246.321,E2 -1246.321} C_VEL
LIN {X 0,Y 594.372,Z 205.445,A -85,B 0,C 180,E1 -1249.095,E2 -1249.095} C_VEL
LIN {X 0,Y 594.413,Z 205.44,A -85,B 0,C 180,E1 -1251.843,E2 -1251.843} C_VEL
LIN {X 0,Y 594.372,Z 205.441,A -85,B 0,C 180,E1 -1254.572,E2 -1254.572} C_VEL
LIN {X 0,Y 594.406,Z 205.445,A -85,B 0,C 180,E1 -1257.289,E2 -1257.289} C_VEL
LIN {X 0,Y 594.414,Z 205.438,A -85,B 0,C 180,E1 -1260,E2 -1260} C_VEL
LIN {X 0,Y 594.386,Z 205.44,A -85,B 0,C 180,E1 -1262.711,E2 -1262.711} C_VEL
LIN {X 0,Y 594.393,Z 205.45,A -85,B 0,C 180,E1 -1265.428,E2 -1265.428} C_VEL
LIN {X 0,Y 594.382,Z 205.44,A -85,B 0,C 180,E1 -1268.157,E2 -1268.157} C_VEL
LIN {X 0,Y 594.376,Z 205.445,A -85,B 0,C 180,E1 -1271.066,E2 -1271.066} C_VEL
LIN {X 0,Y 594.381,Z 205.446,A -85,B 0,C 180,E1 -1273.679,E2 -1273.679} C_VEL
LIN {X 0,Y 594.345,Z 205.448,A -85,B 0,C 180,E1 -1275.3,E2 -1275.3} C_VEL
LIN {X 0,Y 593.676,Z 205.532,A -85,B 0,C 180,E1 -1275.866,E2 -1275.866} C_VEL
LIN {X 0,Y 590.813,Z 205.887,A -85,B 0,C 180,E1 -1276.784,E2 -1276.784} C_VEL
LIN {X 0,Y 588.4,Z 206.193,A -85,B 0,C 180,E1 -1277.522,E2 -1277.522} C_VEL
LIN {X 0,Y 587.373,Z 206.314,A -85,B 0,C 180,E1 -1278.092,E2 -1278.092} C_VEL
LIN {X 0,Y 587.294,Z 206.322,A -85,B 0,C 180,E1 -1278.285,E2 -1278.285} C_VEL
LIN {X 0,Y 587.333,Z 206.322,A -85,B 0,C 180,E1 -1281.038,E2 -1281.038} C_VEL
LIN {X 0,Y 587.321,Z 206.321,A -85,B 0,C 180,E1 -1284.007,E2 -1284.007} C_VEL
LIN {X 0,Y 587.308,Z 206.321,A -85,B 0,C 180,E1 -1286.28,E2 -1286.28} C_VEL
LIN {X 0,Y 587.345,Z 206.322,A -85,B 0,C 180,E1 -1289.132,E2 -1289.132} C_VEL
LIN {X 0,Y 587.341,Z 206.321,A -85,B 0,C 180,E1 -1291.835,E2 -1291.835} C_VEL
LIN {X 0,Y 587.342,Z 206.317,A -85,B 0,C 180,E1 -1294.347,E2 -1294.347} C_VEL
LIN {X 0,Y 587.344,Z 206.324,A -85,B 0,C 180,E1 -1297.608,E2 -1297.608} C_VEL
LIN {X 0,Y 587.309,Z 206.321,A -85,B 0,C 180,E1 -1300.255,E2 -1300.255} C_VEL
LIN {X 0,Y 587.304,Z 206.328,A -85,B 0,C 180,E1 -1303.117,E2 -1303.117} C_VEL
LIN {X 0,Y 587.301,Z 206.323,A -85,B 0,C 180,E1 -1306.047,E2 -1306.047} C_VEL
LIN {X 0,Y 587.333,Z 206.322,A -85,B 0,C 180,E1 -1308.926,E2 -1308.926} C_VEL
LIN {X 0,Y 587.328,Z 206.328,A -85,B 0,C 180,E1 -1311.52,E2 -1311.52} C_VEL
LIN {X 0,Y 587.296,Z 206.323,A -85,B 0,C 180,E1 -1314.463,E2 -1314.463} C_VEL
LIN {X 0,Y 587.339,Z 206.32,A -85,B 0,C 180,E1 -1316.889,E2 -1316.889} C_VEL
LIN {X 0,Y 587.333,Z 206.321,A -85,B 0,C 180,E1 -1319.83,E2 -1319.83} C_VEL
LIN {X 0,Y 587.304,Z 206.322,A -85,B 0,C 180,E1 -1322.317,E2 -1322.317} C_VEL
LIN {X 0,Y 587.333,Z 206.412,A -85,B 0,C 180,E1 -1324.46,E2 -1324.46} C_VEL
LIN {X 0,Y 587.487,Z 215.303,A -85,B 0,C 180,E1 -1326,E2 -1326} C_VEL
LIN {X 0,Y 587.396,Z 230.536,A -85,B 0,C 180,E1 -1328.598,E2 -1328.598} C_VEL
LIN {X 0,Y 587.333,Z 242.136,A -85,B 0,C 180,E1 -1330.554,E2 -1330.554} C_VEL
LIN {X 0,Y 587.857,Z 247.117,A -85,B 0,C 180,E1 -1330.637,E2 -1330.637} C_VEL
LIN {X 0,Y 587.702,Z 349.377,A -85,B 0,C 180,E1 -1331.908,E2 -1331.908} C_VEL
LIN {X 0,Y 587.637,Z 362.776,A -85,B 0,C 180,E1 -1332.221,E2 -1332.221} C_VEL
LIN {X 0,Y 587.613,Z 374.939,A -85,B 0,C 180,E1 -1332.642,E2 -1332.642} C_VEL
LIN {X 0,Y 587.558,Z 386.298,A -85,B 0,C 180,E1 -1333.168,E2 -1333.168} C_VEL
LIN {X 0,Y 587.473,Z 397.744,A -85,B 0,C 180,E1 -1333.851,E2 -1333.851} C_VEL
LIN {X 0,Y 587.375,Z 408.436,A -85,B 0,C 180,E1 -1334.649,E2 -1334.649} C_VEL
LIN {X 0,Y 587.327,Z 418.317,A -85,B 0,C 180,E1 -1335.566,E2 -1335.566} C_VEL
LIN {X 0,Y 587.272,Z 426.524,A -85,B 0,C 180,E1 -1336.505,E2 -1336.505} C_VEL
LIN {X 0,Y 587.219,Z 434.017,A -85,B 0,C 180,E1 -1337.559,E2 -1337.559} C_VEL
LIN {X 0,Y 587.219,Z 439.994,A -85,B 0,C 180,E1 -1338.611,E2 -1338.611} C_VEL
LIN {X 0,Y 587.17,Z 444.678,A -85,B 0,C 180,E1 -1339.657,E2 -1339.657} C_VEL
LIN {X 0,Y 587.173,Z 448.226,A -85,B 0,C 180,E1 -1340.701,E2 -1340.701} C_VEL
LIN {X 0,Y 587.141,Z 450.745,A -85,B 0,C 180,E1 -1341.742,E2 -1341.742} C_VEL
LIN {X 0,Y 587.146,Z 451.907,A -85,B 0,C 180,E1 -1342.434,E2 -1342.434} C_VEL
LIN {X 0,Y 587.188,Z 452.83,A -85,B 0,C 180,E1 -1343.426,E2 -1343.426} C_VEL
LIN {X 0,Y 587.168,Z 452.901,A -85,B 0,C 180,E1 -1344.505,E2 -1344.505} C_VEL
LIN {X 0,Y 587.124,Z 452.439,A -85,B 0,C 180,E1 -1345.193,E2 -1345.193} C_VEL
LIN {X 0,Y 587.17,Z 451.557,A -85,B 0,C 180,E1 -1345.882,E2 -1345.882} C_VEL
LIN {X 0,Y 587.182,Z 450.284,A -85,B 0,C 180,E1 -1346.569,E2 -1346.569} C_VEL
LIN {X 0,Y 587.171,Z 447.578,A -85,B 0,C 180,E1 -1347.599,E2 -1347.599} C_VEL
LIN {X 0,Y 587.161,Z 443.872,A -85,B 0,C 180,E1 -1348.628,E2 -1348.628} C_VEL
LIN {X 0,Y 587.232,Z 439.06,A -85,B 0,C 180,E1 -1349.657,E2 -1349.657} C_VEL
LIN {X 0,Y 587.227,Z 433.011,A -85,B 0,C 180,E1 -1350.686,E2 -1350.686} C_VEL
LIN {X 0,Y 587.305,Z 425.505,A -85,B 0,C 180,E1 -1351.714,E2 -1351.714} C_VEL
LIN {X 0,Y 587.297,Z 417.869,A -85,B 0,C 180,E1 -1352.572,E2 -1352.572} C_VEL
LIN {X 0,Y 587.404,Z 407.52,A -85,B 0,C 180,E1 -1353.515,E2 -1353.515} C_VEL
LIN {X 0,Y 587.448,Z 397.027,A -85,B 0,C 180,E1 -1354.288,E2 -1354.288} C_VEL
LIN {X 0,Y 587.558,Z 385.255,A -85,B 0,C 180,E1 -1354.975,E2 -1354.975} C_VEL
LIN {X 0,Y 587.601,Z 372.744,A -85,B 0,C 180,E1 -1355.534,E2 -1355.534} C_VEL
LIN {X 0,Y 587.657,Z 360.228,A -85,B 0,C 180,E1 -1355.942,E2 -1355.942} C_VEL
LIN {X 0,Y 587.721,Z 347.748,A -85,B 0,C 180,E1 -1356.21,E2 -1356.21} C_VEL
LIN {X 0,Y 587.758,Z 244.902,A -85,B 0,C 180,E1 -1357.482,E2 -1357.482} C_VEL
LIN {X 0,Y 587.333,Z 242.099,A -85,B 0,C 180,E1 -1357.542,E2 -1357.542} C_VEL
LIN {X 0,Y 587.453,Z 225.551,A -85,B 0,C 180,E1 -1360.338,E2 -1360.338} C_VEL
LIN {X 0,Y 587.538,Z 208.205,A -85,B 0,C 180,E1 -1363.313,E2 -1363.313} C_VEL
LIN {X 0,Y 587.333,Z 206.323,A -85,B 0,C 180,E1 -1363.67,E2 -1363.67} C_VEL
LIN {X 0,Y 587.363,Z 206.324,A -85,B 0,C 180,E1 -1366.817,E2 -1366.817} C_VEL
LIN {X 0,Y 587.313,Z 206.321,A -85,B 0,C 180,E1 -1369.576,E2 -1369.576} C_VEL
LIN {X 0,Y 587.321,Z 206.32,A -85,B 0,C 180,E1 -1371.774,E2 -1371.774} C_VEL
LIN {X 0,Y 587.35,Z 206.326,A -85,B 0,C 180,E1 -1374.759,E2 -1374.759} C_VEL
LIN {X 0,Y 587.313,Z 206.325,A -85,B 0,C 180,E1 -1377.047,E2 -1377.047} C_VEL
LIN {X 0,Y 587.345,Z 206.318,A -85,B 0,C 180,E1 -1379.38,E2 -1379.38} C_VEL
LIN {X 0,Y 587.344,Z 206.317,A -85,B 0,C 180,E1 -1381.835,E2 -1381.835} C_VEL
LIN {X 0,Y 587.346,Z 206.321,A -85,B 0,C 180,E1 -1384.347,E2 -1384.347} C_VEL
LIN {X 0,Y 587.344,Z 206.317,A -85,B 0,C 180,E1 -1387.608,E2 -1387.608} C_VEL
LIN {X 0,Y 587.312,Z 206.324,A -85,B 0,C 180,E1 -1390.254,E2 -1390.254} C_VEL
LIN {X 0,Y 587.305,Z 206.325,A -85,B 0,C 180,E1 -1393.117,E2 -1393.117} C_VEL
LIN {X 0,Y 587.315,Z 206.322,A -85,B 0,C 180,E1 -1396.048,E2 -1396.048} C_VEL
LIN {X 0,Y 587.335,Z 206.324,A -85,B 0,C 180,E1 -1398.925,E2 -1398.925} C_VEL
LIN {X 0,Y 587.321,Z 206.32,A -85,B 0,C 180,E1 -1401.52,E2 -1401.52} C_VEL
LIN {X 0,Y 587.29,Z 206.326,A -85,B 0,C 180,E1 -1404.1,E2 -1404.1} C_VEL
LIN {X 0,Y 587.335,Z 206.328,A -85,B 0,C 180,E1 -1406.603,E2 -1406.603} C_VEL
LIN {X 0,Y 587.336,Z 206.318,A -85,B 0,C 180,E1 -1409.49,E2 -1409.49} C_VEL
LIN {X 0,Y 587.342,Z 206.322,A -85,B 0,C 180,E1 -1412.309,E2 -1412.309} C_VEL
LIN {X 0,Y 587.341,Z 206.318,A -85,B 0,C 180,E1 -1415.423,E2 -1415.423} C_VEL
LIN {X 0,Y 587.316,Z 206.324,A -85,B 0,C 180,E1 -1418.225,E2 -1418.225} C_VEL
LIN {X 0,Y 587.341,Z 206.32,A -85,B 0,C 180,E1 -1421.151,E2 -1421.151} C_VEL
LIN {X 0,Y 587.321,Z 206.321,A -85,B 0,C 180,E1 -1423.31,E2 -1423.31} C_VEL
LIN {X 0,Y 587.359,Z 206.318,A -85,B 0,C 180,E1 -1426.154,E2 -1426.154} C_VEL
LIN {X 0,Y 587.338,Z 206.322,A -85,B 0,C 180,E1 -1428.962,E2 -1428.962} C_VEL
LIN {X 0,Y 587.341,Z 206.317,A -85,B 0,C 180,E1 -1431.744,E2 -1431.744} C_VEL
LIN {X 0,Y 587.362,Z 206.323,A -85,B 0,C 180,E1 -1434.507,E2 -1434.507} C_VEL
LIN {X 0,Y 587.357,Z 206.316,A -85,B 0,C 180,E1 -1437.257,E2 -1437.257} C_VEL
LIN {X 0,Y 587.383,Z 206.313,A -85,B 0,C 180,E1 -1440,E2 -1440} C_VEL
LIN {X 0,Y 587.374,Z 206.321,A -85,B 0,C 180,E1 -1442.743,E2 -1442.743} C_VEL
LIN {X 0,Y 587.342,Z 206.317,A -85,B 0,C 180,E1 -1445.493,E2 -1445.493} C_VEL
LIN {X 0,Y 587.365,Z 206.319,A -85,B 0,C 180,E1 -1448.255,E2 -1448.255} C_VEL
LIN {X 0,Y 587.35,Z 206.318,A -85,B 0,C 180,E1 -1451.134,E2 -1451.134} C_VEL
LIN {X 0,Y 587.366,Z 206.319,A -85,B 0,C 180,E1 -1454.26,E2 -1454.26} C_VEL
LIN {X 0,Y 587.313,Z 206.321,A -85,B 0,C 180,E1 -1457.407,E2 -1457.407} C_VEL
LIN {X 0,Y 587.31,Z 206.321,A -85,B 0,C 180,E1 -1459.576,E2 -1459.576} C_VEL
LIN {X 0,Y 587.317,Z 206.32,A -85,B 0,C 180,E1 -1461.775,E2 -1461.775} C_VEL
LIN {X 0,Y 587.346,Z 206.324,A -85,B 0,C 180,E1 -1464.759,E2 -1464.759} C_VEL
LIN {X 0,Y 587.302,Z 206.325,A -85,B 0,C 180,E1 -1467.048,E2 -1467.048} C_VEL
LIN {X 0,Y 587.342,Z 206.317,A -85,B 0,C 180,E1 -1469.38,E2 -1469.38} C_VEL
LIN {X 0,Y 587.342,Z 206.318,A -85,B 0,C 180,E1 -1471.835,E2 -1471.835} C_VEL
LIN {X 0,Y 587.341,Z 206.324,A -85,B 0,C 180,E1 -1474.347,E2 -1474.347} C_VEL
LIN {X 0,Y 587.341,Z 206.317,A -85,B 0,C 180,E1 -1477.608,E2 -1477.608} C_VEL
LIN {X 0,Y 587.31,Z 206.326,A -85,B 0,C 180,E1 -1480.255,E2 -1480.255} C_VEL
LIN {X 0,Y 587.303,Z 206.324,A -85,B 0,C 180,E1 -1483.117,E2 -1483.117} C_VEL
LIN {X 0,Y 587.313,Z 206.323,A -85,B 0,C 180,E1 -1486.049,E2 -1486.049} C_VEL
LIN {X 0,Y 587.333,Z 206.322,A -85,B 0,C 180,E1 -1488.926,E2 -1488.926} C_VEL
LIN {X 0,Y 587.318,Z 206.32,A -85,B 0,C 180,E1 -1491.52,E2 -1491.52} C_VEL
LIN {X 0,Y 587.289,Z 206.327,A -85,B 0,C 180,E1 -1494.1,E2 -1494.1} C_VEL
LIN {X 0,Y 587.335,Z 206.327,A -85,B 0,C 180,E1 -1496.603,E2 -1496.603} C_VEL
LIN {X 0,Y 587.322,Z 206.319,A -85,B 0,C 180,E1 -1499.493,E2 -1499.493} C_VEL
LIN {X 0,Y 587.342,Z 206.324,A -85,B 0,C 180,E1 -1502.309,E2 -1502.309} C_VEL
LIN {X 0,Y 587.341,Z 206.318,A -85,B 0,C 180,E1 -1505.423,E2 -1505.423} C_VEL
LIN {X 0,Y 587.332,Z 206.463,A -85,B 0,C 180,E1 -1507.262,E2 -1507.262} C_VEL
LIN {X 0,Y 587.834,Z 210.502,A -85,B 0,C 180,E1 -1507.876,E2 -1507.876} C_VEL
LIN {X 0,Y 587.663,Z 230.067,A -85,B 0,C 180,E1 -1510.715,E2 -1510.715} C_VEL
LIN {X 0,Y 587.521,Z 249.541,A -85,B 0,C 180,E1 -1513.495,E2 -1513.495} C_VEL
LIN {X 0,Y 587.427,Z 269.691,A -85,B 0,C 180,E1 -1516.332,E2 -1516.332} C_VEL
LIN {X 0,Y 587.423,Z 271.144,A -85,B 0,C 180,E1 -1516.509,E2 -1516.509} C_VEL
LIN {X 0,Y 587.84,Z 276.51,A -85,B 0,C 180,E1 -1516.584,E2 -1516.584} C_VEL
LIN {X 0,Y 587.724,Z 378.948,A -85,B 0,C 180,E1 -1517.855,E2 -1517.855} C_VEL
LIN {X 0,Y 587.677,Z 392.22,A -85,B 0,C 180,E1 -1518.161,E2 -1518.161} C_VEL
LIN {X 0,Y 587.597,Z 404.778,A -85,B 0,C 180,E1 -1518.59,E2 -1518.59} C_VEL
LIN {X 0,Y 587.551,Z 416.63,A -85,B 0,C 180,E1 -1519.141,E2 -1519.141} C_VEL
LIN {X 0,Y 587.454,Z 428.203,A -85,B 0,C 180,E1 -1519.836,E2 -1519.836} C_VEL
LIN {X 0,Y 587.393,Z 438.599,A -85,B 0,C 180,E1 -1520.618,E2 -1520.618} C_VEL
LIN {X 0,Y 587.321,Z 447.113,A -85,B 0,C 180,E1 -1521.398,E2 -1521.398} C_VEL
LIN {X 0,Y 587.274,Z 454.961,A -85,B 0,C 180,E1 -1522.263,E2 -1522.263} C_VEL
LIN {X 0,Y 587.23,Z 461.469,A -85,B 0,C 180,E1 -1523.126,E2 -1523.126} C_VEL
LIN {X 0,Y 587.236,Z 467.867,A -85,B 0,C 180,E1 -1524.161,E2 -1524.161} C_VEL
LIN {X 0,Y 587.147,Z 472.95,A -85,B 0,C 180,E1 -1525.194,E2 -1525.194} C_VEL
LIN {X 0,Y 587.213,Z 476.896,A -85,B 0,C 180,E1 -1526.226,E2 -1526.226} C_VEL
LIN {X 0,Y 587.132,Z 479.809,A -85,B 0,C 180,E1 -1527.256,E2 -1527.256} C_VEL
LIN {X 0,Y 587.14,Z 481.2,A -85,B 0,C 180,E1 -1527.942,E2 -1527.942} C_VEL
LIN {X 0,Y 587.14,Z 482.784,A -85,B 0,C 180,E1 -1529.314,E2 -1529.314} C_VEL
LIN {X 0,Y 587.137,Z 483,A -85,B 0,C 180,E1 -1530,E2 -1530} C_VEL
LIN {X 0,Y 587.147,Z 482.186,A -85,B 0,C 180,E1 -1531.372,E2 -1531.372} C_VEL
LIN {X 0,Y 587.14,Z 481.201,A -85,B 0,C 180,E1 -1532.058,E2 -1532.058} C_VEL
LIN {X 0,Y 587.132,Z 479.81,A -85,B 0,C 180,E1 -1532.744,E2 -1532.744} C_VEL
LIN {X 0,Y 587.213,Z 476.896,A -85,B 0,C 180,E1 -1533.774,E2 -1533.774} C_VEL
LIN {X 0,Y 587.147,Z 472.949,A -85,B 0,C 180,E1 -1534.806,E2 -1534.806} C_VEL
LIN {X 0,Y 587.217,Z 466.877,A -85,B 0,C 180,E1 -1536.011,E2 -1536.011} C_VEL
LIN {X 0,Y 587.245,Z 460.237,A -85,B 0,C 180,E1 -1537.046,E2 -1537.046} C_VEL
LIN {X 0,Y 587.3,Z 451.99,A -85,B 0,C 180,E1 -1538.083,E2 -1538.083} C_VEL
LIN {X 0,Y 587.343,Z 443.538,A -85,B 0,C 180,E1 -1538.949,E2 -1538.949} C_VEL
LIN {X 0,Y 587.418,Z 433.096,A -85,B 0,C 180,E1 -1539.816,E2 -1539.816} C_VEL
LIN {X 0,Y 587.508,Z 422.756,A -85,B 0,C 180,E1 -1540.511,E2 -1540.511} C_VEL
LIN {X 0,Y 587.568,Z 410.978,A -85,B 0,C 180,E1 -1541.141,E2 -1541.141} C_VEL
LIN {X 0,Y 587.61,Z 398.596,A -85,B 0,C 180,E1 -1541.64,E2 -1541.64} C_VEL
LIN {X 0,Y 587.69,Z 385.434,A -85,B 0,C 180,E1 -1542.014,E2 -1542.014} C_VEL
LIN {X 0,Y 587.718,Z 373.082,A -85,B 0,C 180,E1 -1542.233,E2 -1542.233} C_VEL
LIN {X 0,Y 587.701,Z 272.929,A -85,B 0,C 180,E1 -1543.463,E2 -1543.463} C_VEL
LIN {X 0,Y 587.379,Z 270.792,A -85,B 0,C 180,E1 -1543.515,E2 -1543.515} C_VEL
LIN {X 0,Y 587.481,Z 253.319,A -85,B 0,C 180,E1 -1545.971,E2 -1545.971} C_VEL
LIN {X 0,Y 587.596,Z 235.688,A -85,B 0,C 180,E1 -1548.479,E2 -1548.479} C_VEL
LIN {X 0,Y 587.721,Z 218.058,A -85,B 0,C 180,E1 -1551.023,E2 -1551.023} C_VEL
LIN {X 0,Y 587.813,Z 209.242,A -85,B 0,C 180,E1 -1552.309,E2 -1552.309} C_VEL
LIN {X 0,Y 587.319,Z 206.327,A -85,B 0,C 180,E1 -1552.788,E2 -1552.788} C_VEL
LIN {X 0,Y 587.331,Z 206.329,A -85,B 0,C 180,E1 -1555.517,E2 -1555.517} C_VEL
LIN {X 0,Y 587.338,Z 206.323,A -85,B 0,C 180,E1 -1557.818,E2 -1557.818} C_VEL
LIN {X 0,Y 587.322,Z 206.32,A -85,B 0,C 180,E1 -1560.507,E2 -1560.507} C_VEL
LIN {X 0,Y 587.335,Z 206.328,A -85,B 0,C 180,E1 -1563.397,E2 -1563.397} C_VEL
LIN {X 0,Y 587.289,Z 206.327,A -85,B 0,C 180,E1 -1565.9,E2 -1565.9} C_VEL
LIN {X 0,Y 587.319,Z 206.32,A -85,B 0,C 180,E1 -1568.48,E2 -1568.48} C_VEL
LIN {X 0,Y 587.334,Z 206.323,A -85,B 0,C 180,E1 -1571.157,E2 -1571.157} C_VEL
LIN {X 0,Y 587.313,Z 206.322,A -85,B 0,C 180,E1 -1574.112,E2 -1574.112} C_VEL
LIN {X 0,Y 587.304,Z 206.325,A -85,B 0,C 180,E1 -1576.992,E2 -1576.992} C_VEL
LIN {X 0,Y 587.311,Z 206.326,A -85,B 0,C 180,E1 -1579.745,E2 -1579.745} C_VEL
LIN {X 0,Y 587.322,Z 206.319,A -85,B 0,C 180,E1 -1582.39,E2 -1582.39} C_VEL
LIN {X 0,Y 587.341,Z 206.324,A -85,B 0,C 180,E1 -1585.653,E2 -1585.653} C_VEL
LIN {X 0,Y 587.339,Z 206.318,A -85,B 0,C 180,E1 -1588.231,E2 -1588.231} C_VEL
LIN {X 0,Y 587.346,Z 206.318,A -85,B 0,C 180,E1 -1590.867,E2 -1590.867} C_VEL
LIN {X 0,Y 587.336,Z 206.321,A -85,B 0,C 180,E1 -1593.824,E2 -1593.824} C_VEL
LIN {X 0,Y 587.329,Z 206.321,A -85,B 0,C 180,E1 -1595.993,E2 -1595.993} C_VEL
LIN {X 0,Y 587.317,Z 206.32,A -85,B 0,C 180,E1 -1598.225,E2 -1598.225} C_VEL
LIN {X 0,Y 587.349,Z 206.322,A -85,B 0,C 180,E1 -1601.151,E2 -1601.151} C_VEL
LIN {X 0,Y 587.314,Z 206.322,A -85,B 0,C 180,E1 -1604.025,E2 -1604.025} C_VEL
LIN {X 0,Y 587.354,Z 206.316,A -85,B 0,C 180,E1 -1606.154,E2 -1606.154} C_VEL
LIN {X 0,Y 587.339,Z 206.32,A -85,B 0,C 180,E1 -1608.962,E2 -1608.962} C_VEL
LIN {X 0,Y 587.365,Z 206.319,A -85,B 0,C 180,E1 -1611.745,E2 -1611.745} C_VEL
LIN {X 0,Y 587.34,Z 206.317,A -85,B 0,C 180,E1 -1614.507,E2 -1614.507} C_VEL
LIN {X 0,Y 587.37,Z 206.321,A -85,B 0,C 180,E1 -1617.257,E2 -1617.257} C_VEL
LIN {X 0,Y 587.383,Z 206.314,A -85,B 0,C 180,E1 -1620,E2 -1620} C_VEL
LIN {X 0,Y 587.355,Z 206.316,A -85,B 0,C 180,E1 -1622.743,E2 -1622.743} C_VEL
LIN {X 0,Y 587.359,Z 206.324,A -85,B 0,C 180,E1 -1625.493,E2 -1625.493} C_VEL
LIN {X 0,Y 587.341,Z 206.317,A -85,B 0,C 180,E1 -1628.256,E2 -1628.256} C_VEL
LIN {X 0,Y 587.35,Z 206.321,A -85,B 0,C 180,E1 -1631.134,E2 -1631.134} C_VEL
LIN {X 0,Y 587.342,Z 206.317,A -85,B 0,C 180,E1 -1634.251,E2 -1634.251} C_VEL
LIN {X 0,Y 587.34,Z 206.327,A -85,B 0,C 180,E1 -1637.406,E2 -1637.406} C_VEL
LIN {X 0,Y 587.294,Z 206.322,A -85,B 0,C 180,E1 -1638.285,E2 -1638.285} C_VEL
LIN {X 0,Y 586.653,Z 206.405,A -85,B 0,C 180,E1 -1638.857,E2 -1638.857} C_VEL
LIN {X 0,Y 583.845,Z 206.757,A -85,B 0,C 180,E1 -1639.786,E2 -1639.786} C_VEL
LIN {X 0,Y 581.444,Z 207.054,A -85,B 0,C 180,E1 -1640.533,E2 -1640.533} C_VEL
LIN {X 0,Y 580.386,Z 207.189,A -85,B 0,C 180,E1 -1641.11,E2 -1641.11} C_VEL
LIN {X 0,Y 580.285,Z 207.205,A -85,B 0,C 180,E1 -1641.305,E2 -1641.305} C_VEL
LIN {X 0,Y 580.288,Z 207.196,A -85,B 0,C 180,E1 -1644.317,E2 -1644.317} C_VEL
LIN {X 0,Y 580.28,Z 207.207,A -85,B 0,C 180,E1 -1647.402,E2 -1647.402} C_VEL
LIN {X 0,Y 580.278,Z 207.201,A -85,B 0,C 180,E1 -1649.773,E2 -1649.773} C_VEL
LIN {X 0,Y 580.296,Z 207.195,A -85,B 0,C 180,E1 -1652.201,E2 -1652.201} C_VEL
LIN {X 0,Y 580.287,Z 207.197,A -85,B 0,C 180,E1 -1654.697,E2 -1654.697} C_VEL
LIN {X 0,Y 580.289,Z 207.203,A -85,B 0,C 180,E1 -1657.269,E2 -1657.269} C_VEL
LIN {X 0,Y 580.289,Z 207.196,A -85,B 0,C 180,E1 -1660.27,E2 -1660.27} C_VEL
LIN {X 0,Y 580.269,Z 207.199,A -85,B 0,C 180,E1 -1662.707,E2 -1662.707} C_VEL
LIN {X 0,Y 580.252,Z 207.207,A -85,B 0,C 180,E1 -1665.611,E2 -1665.611} C_VEL
LIN {X 0,Y 580.28,Z 207.198,A -85,B 0,C 180,E1 -1668.231,E2 -1668.231} C_VEL
LIN {X 0,Y 580.275,Z 207.201,A -85,B 0,C 180,E1 -1670.965,E2 -1670.965} C_VEL
LIN {X 0,Y 580.252,Z 207.208,A -85,B 0,C 180,E1 -1673.595,E2 -1673.595} C_VEL
LIN {X 0,Y 580.312,Z 207.194,A -85,B 0,C 180,E1 -1676.145,E2 -1676.145} C_VEL
LIN {X 0,Y 580.275,Z 207.198,A -85,B 0,C 180,E1 -1678.614,E2 -1678.614} C_VEL
LIN {X 0,Y 580.292,Z 207.199,A -85,B 0,C 180,E1 -1681.024,E2 -1681.024} C_VEL
LIN {X 0,Y 580.288,Z 207.199,A -85,B 0,C 180,E1 -1684.151,E2 -1684.151} C_VEL
LIN {X 0,Y 580.323,Z 207.436,A -85,B 0,C 180,E1 -1684.393,E2 -1684.393} C_VEL
LIN {X 0,Y 580.487,Z 214.828,A -85,B 0,C 180,E1 -1685.692,E2 -1685.692} C_VEL
LIN {X 0,Y 580.368,Z 228.979,A -85,B 0,C 180,E1 -1688.138,E2 -1688.138} C_VEL
LIN {X 0,Y 580.312,Z 242.16,A -85,B 0,C 180,E1 -1690.392,E2 -1690.392} C_VEL
LIN {X 0,Y 580.964,Z 246.98,A -85,B 0,C 180,E1 -1690.473,E2 -1690.473} C_VEL
LIN {X 0,Y 580.764,Z 348.962,A -85,B 0,C 180,E1 -1691.753,E2 -1691.753} C_VEL
LIN {X 0,Y 580.698,Z 362.502,A -85,B 0,C 180,E1 -1692.07,E2 -1692.07} C_VEL
LIN {X 0,Y 580.654,Z 374.513,A -85,B 0,C 180,E1 -1692.487,E2 -1692.487} C_VEL
LIN {X 0,Y 580.571,Z 385.702,A -85,B 0,C 180,E1 -1693.004,E2 -1693.004} C_VEL
LIN {X 0,Y 580.475,Z 396.631,A -85,B 0,C 180,E1 -1693.651,E2 -1693.651} C_VEL
LIN {X 0,Y 580.379,Z 407.529,A -85,B 0,C 180,E1 -1694.46,E2 -1694.46} C_VEL
LIN {X 0,Y 580.293,Z 417.878,A -85,B 0,C 180,E1 -1695.415,E2 -1695.415} C_VEL
LIN {X 0,Y 580.22,Z 425.943,A -85,B 0,C 180,E1 -1696.338,E2 -1696.338} C_VEL
LIN {X 0,Y 580.17,Z 433.541,A -85,B 0,C 180,E1 -1697.406,E2 -1697.406} C_VEL
LIN {X 0,Y 580.123,Z 439.607,A -85,B 0,C 180,E1 -1698.469,E2 -1698.469} C_VEL
LIN {X 0,Y 580.091,Z 444.376,A -85,B 0,C 180,E1 -1699.529,E2 -1699.529} C_VEL
LIN {X 0,Y 580.073,Z 448.002,A -85,B 0,C 180,E1 -1700.586,E2 -1700.586} C_VEL
LIN {X 0,Y 580.062,Z 450.594,A -85,B 0,C 180,E1 -1701.64,E2 -1701.64} C_VEL
LIN {X 0,Y 580.066,Z 451.804,A -85,B 0,C 180,E1 -1702.341,E2 -1702.341} C_VEL
LIN {X 0,Y 580.1,Z 452.843,A -85,B 0,C 180,E1 -1703.438,E2 -1703.438} C_VEL
LIN {X 0,Y 580.089,Z 452.917,A -85,B 0,C 180,E1 -1704.438,E2 -1704.438} C_VEL
LIN {X 0,Y 580.028,Z 452.512,A -85,B 0,C 180,E1 -1705.134,E2 -1705.134} C_VEL
LIN {X 0,Y 580.087,Z 451.672,A -85,B 0,C 180,E1 -1705.831,E2 -1705.831} C_VEL
LIN {X 0,Y 580.108,Z 450.434,A -85,B 0,C 180,E1 -1706.527,E2 -1706.527} C_VEL
LIN {X 0,Y 580.09,Z 447.8,A -85,B 0,C 180,E1 -1707.57,E2 -1707.57} C_VEL
LIN {X 0,Y 580.066,Z 444.17,A -85,B 0,C 180,E1 -1708.611,E2 -1708.611} C_VEL
LIN {X 0,Y 580.141,Z 439.439,A -85,B 0,C 180,E1 -1709.653,E2 -1709.653} C_VEL
LIN {X 0,Y 580.189,Z 432.365,A -85,B 0,C 180,E1 -1710.868,E2 -1710.868} C_VEL
LIN {X 0,Y 580.268,Z 424.688,A -85,B 0,C 180,E1 -1711.909,E2 -1711.909} C_VEL
LIN {X 0,Y 580.296,Z 415.108,A -85,B 0,C 180,E1 -1712.95,E2 -1712.95} C_VEL
LIN {X 0,Y 580.41,Z 405.232,A -85,B 0,C 180,E1 -1713.819,E2 -1713.819} C_VEL
LIN {X 0,Y 580.49,Z 394.109,A -85,B 0,C 180,E1 -1714.601,E2 -1714.601} C_VEL
LIN {X 0,Y 580.603,Z 383.247,A -85,B 0,C 180,E1 -1715.209,E2 -1715.209} C_VEL
LIN {X 0,Y 580.641,Z 371.274,A -85,B 0,C 180,E1 -1715.731,E2 -1715.731} C_VEL
LIN {X 0,Y 580.767,Z 358.86,A -85,B 0,C 180,E1 -1716.122,E2 -1716.122} C_VEL
LIN {X 0,Y 580.808,Z 345.393,A -85,B 0,C 180,E1 -1716.392,E2 -1716.392} C_VEL
LIN {X 0,Y 580.908,Z 245.921,A -85,B 0,C 180,E1 -1717.631,E2 -1717.631} C_VEL
LIN {X 0,Y 580.3,Z 242.152,A -85,B 0,C 180,E1 -1717.699,E2 -1717.699} C_VEL
LIN {X 0,Y 580.457,Z 225.992,A -85,B 0,C 180,E1 -1720.464,E2 -1720.464} C_VEL
LIN {X 0,Y 580.549,Z 209.667,A -85,B 0,C 180,E1 -1723.298,E2 -1723.298} C_VEL
LIN {X 0,Y 580.303,Z 207.199,A -85,B 0,C 180,E1 -1723.749,E2 -1723.749} C_VEL
LIN {X 0,Y 580.277,Z 207.201,A -85,B 0,C 180,E1 -1726.174,E2 -1726.174} C_VEL
LIN {X 0,Y 580.3,Z 207.198,A -85,B 0,C 180,E1 -1729.087,E2 -1729.087} C_VEL
LIN {X 0,Y 580.272,Z 207.199,A -85,B 0,C 180,E1 -1732.053,E2 -1732.053} C_VEL
LIN {X 0,Y 580.303,Z 207.198,A -85,B 0,C 180,E1 -1735.08,E2 -1735.08} C_VEL
LIN {X 0,Y 580.284,Z 207.199,A -85,B 0,C 180,E1 -1738.186,E2 -1738.186} C_VEL
LIN {X 0,Y 580.285,Z 207.207,A -85,B 0,C 180,E1 -1740.694,E2 -1740.694} C_VEL
LIN {X 0,Y 580.286,Z 207.197,A -85,B 0,C 180,E1 -1743.313,E2 -1743.313} C_VEL
LIN {X 0,Y 580.247,Z 207.201,A -85,B 0,C 180,E1 -1745.756,E2 -1745.756} C_VEL
LIN {X 0,Y 580.289,Z 207.198,A -85,B 0,C 180,E1 -1748.146,E2 -1748.146} C_VEL
LIN {X 0,Y 580.297,Z 207.202,A -85,B 0,C 180,E1 -1750.844,E2 -1750.844} C_VEL
LIN {X 0,Y 580.27,Z 207.198,A -85,B 0,C 180,E1 -1753.659,E2 -1753.659} C_VEL
LIN {X 0,Y 580.269,Z 207.208,A -85,B 0,C 180,E1 -1756.61,E2 -1756.61} C_VEL
LIN {X 0,Y 580.298,Z 207.197,A -85,B 0,C 180,E1 -1759.156,E2 -1759.156} C_VEL
LIN {X 0,Y 580.288,Z 207.196,A -85,B 0,C 180,E1 -1761.927,E2 -1761.927} C_VEL
LIN {X 0,Y 580.25,Z 207.207,A -85,B 0,C 180,E1 -1764.452,E2 -1764.452} C_VEL
LIN {X 0,Y 580.29,Z 207.2,A -85,B 0,C 180,E1 -1766.975,E2 -1766.975} C_VEL
LIN {X 0,Y 580.295,Z 207.195,A -85,B 0,C 180,E1 -1769.425,E2 -1769.425} C_VEL
LIN {X 0,Y 580.29,Z 207.198,A -85,B 0,C 180,E1 -1772.143,E2 -1772.143} C_VEL
LIN {X 0,Y 580.289,Z 207.201,A -85,B 0,C 180,E1 -1774.919,E2 -1774.919} C_VEL
LIN {X 0,Y 580.267,Z 207.199,A -85,B 0,C 180,E1 -1777.947,E2 -1777.947} C_VEL
LIN {X 0,Y 580.292,Z 207.201,A -85,B 0,C 180,E1 -1780.913,E2 -1780.913} C_VEL
LIN {X 0,Y 580.262,Z 207.199,A -85,B 0,C 180,E1 -1783.825,E2 -1783.825} C_VEL
LIN {X 0,Y 580.317,Z 207.193,A -85,B 0,C 180,E1 -1785.983,E2 -1785.983} C_VEL
LIN {X 0,Y 580.307,Z 207.2,A -85,B 0,C 180,E1 -1788.827,E2 -1788.827} C_VEL
LIN {X 0,Y 580.31,Z 207.193,A -85,B 0,C 180,E1 -1791.644,E2 -1791.644} C_VEL
LIN {X 0,Y 580.328,Z 207.198,A -85,B 0,C 180,E1 -1794.44,E2 -1794.44} C_VEL
LIN {X 0,Y 580.325,Z 207.193,A -85,B 0,C 180,E1 -1797.223,E2 -1797.223} C_VEL
LIN {X 0,Y 580.353,Z 207.189,A -85,B 0,C 180,E1 -1800,E2 -1800} C_VEL
LIN {X 0,Y 580.339,Z 207.197,A -85,B 0,C 180,E1 -1802.776,E2 -1802.776} C_VEL
LIN {X 0,Y 580.31,Z 207.193,A -85,B 0,C 180,E1 -1805.56,E2 -1805.56} C_VEL
LIN {X 0,Y 580.317,Z 207.192,A -85,B 0,C 180,E1 -1807.655,E2 -1807.655} C_VEL
LIN {X 0,Y 580.3,Z 207.203,A -85,B 0,C 180,E1 -1810.467,E2 -1810.467} C_VEL
LIN {X 0,Y 580.268,Z 207.199,A -85,B 0,C 180,E1 -1813.304,E2 -1813.304} C_VEL
LIN {X 0,Y 580.288,Z 207.196,A -85,B 0,C 180,E1 -1815.453,E2 -1815.453} C_VEL
LIN {X 0,Y 580.271,Z 207.198,A -85,B 0,C 180,E1 -1817.625,E2 -1817.625} C_VEL
LIN {X 0,Y 580.285,Z 207.197,A -85,B 0,C 180,E1 -1819.823,E2 -1819.823} C_VEL
LIN {X 0,Y 580.268,Z 207.201,A -85,B 0,C 180,E1 -1822.053,E2 -1822.053} C_VEL
LIN {X 0,Y 580.3,Z 207.197,A -85,B 0,C 180,E1 -1825.08,E2 -1825.08} C_VEL
LIN {X 0,Y 580.281,Z 207.201,A -85,B 0,C 180,E1 -1828.187,E2 -1828.187} C_VEL
LIN {X 0,Y 580.281,Z 207.205,A -85,B 0,C 180,E1 -1830.694,E2 -1830.694} C_VEL
LIN {X 0,Y 580.283,Z 207.197,A -85,B 0,C 180,E1 -1833.313,E2 -1833.313} C_VEL
LIN {X 0,Y 580.244,Z 207.202,A -85,B 0,C 180,E1 -1835.756,E2 -1835.756} C_VEL
LIN {X 0,Y 580.287,Z 207.199,A -85,B 0,C 180,E1 -1838.147,E2 -1838.147} C_VEL
LIN {X 0,Y 580.294,Z 207.2,A -85,B 0,C 180,E1 -1840.844,E2 -1840.844} C_VEL
LIN {X 0,Y 580.242,Z 207.202,A -85,B 0,C 180,E1 -1843.662,E2 -1843.662} C_VEL
LIN {X 0,Y 580.267,Z 207.208,A -85,B 0,C 180,E1 -1846.611,E2 -1846.611} C_VEL
LIN {X 0,Y 580.295,Z 207.196,A -85,B 0,C 180,E1 -1849.156,E2 -1849.156} C_VEL
LIN {X 0,Y 580.287,Z 207.197,A -85,B 0,C 180,E1 -1851.928,E2 -1851.928} C_VEL
LIN {X 0,Y 580.249,Z 207.21,A -85,B 0,C 180,E1 -1854.453,E2 -1854.453} C_VEL
LIN {X 0,Y 580.289,Z 207.199,A -85,B 0,C 180,E1 -1856.975,E2 -1856.975} C_VEL
LIN {X 0,Y 580.283,Z 207.196,A -85,B 0,C 180,E1 -1859.424,E2 -1859.424} C_VEL
LIN {X 0,Y 580.289,Z 207.2,A -85,B 0,C 180,E1 -1862.143,E2 -1862.143} C_VEL
LIN {X 0,Y 580.289,Z 207.2,A -85,B 0,C 180,E1 -1864.919,E2 -1864.919} C_VEL
LIN {X 0,Y 580.284,Z 207.226,A -85,B 0,C 180,E1 -1867.107,E2 -1867.107} C_VEL
LIN {X 0,Y 580.908,Z 211.687,A -85,B 0,C 180,E1 -1867.786,E2 -1867.786} C_VEL
LIN {X 0,Y 580.703,Z 230.406,A -85,B 0,C 180,E1 -1870.524,E2 -1870.524} C_VEL
LIN {X 0,Y 580.537,Z 249.541,A -85,B 0,C 180,E1 -1873.291,E2 -1873.291} C_VEL
LIN {X 0,Y 580.389,Z 270.792,A -85,B 0,C 180,E1 -1876.32,E2 -1876.32} C_VEL
LIN {X 0,Y 580.937,Z 276.51,A -85,B 0,C 180,E1 -1876.422,E2 -1876.422} C_VEL
LIN {X 0,Y 580.781,Z 378.947,A -85,B 0,C 180,E1 -1877.708,E2 -1877.708} C_VEL
LIN {X 0,Y 580.735,Z 392.22,A -85,B 0,C 180,E1 -1878.017,E2 -1878.017} C_VEL
LIN {X 0,Y 580.631,Z 404.375,A -85,B 0,C 180,E1 -1878.436,E2 -1878.436} C_VEL
LIN {X 0,Y 580.554,Z 416.629,A -85,B 0,C 180,E1 -1879.008,E2 -1879.008} C_VEL
LIN {X 0,Y 580.428,Z 428.202,A -85,B 0,C 180,E1 -1879.712,E2 -1879.712} C_VEL
LIN {X 0,Y 580.344,Z 438.6,A -85,B 0,C 180,E1 -1880.503,E2 -1880.503} C_VEL
LIN {X 0,Y 580.271,Z 447.113,A -85,B 0,C 180,E1 -1881.292,E2 -1881.292} C_VEL
LIN {X 0,Y 580.222,Z 454.961,A -85,B 0,C 180,E1 -1882.168,E2 -1882.168} C_VEL
LIN {X 0,Y 580.154,Z 462.65,A -85,B 0,C 180,E1 -1883.222,E2 -1883.222} C_VEL
LIN {X 0,Y 580.139,Z 469.68,A -85,B 0,C 180,E1 -1884.438,E2 -1884.438} C_VEL
LIN {X 0,Y 580.108,Z 474.372,A -85,B 0,C 180,E1 -1885.483,E2 -1885.483} C_VEL
LIN {X 0,Y 580.123,Z 477.957,A -85,B 0,C 180,E1 -1886.527,E2 -1886.527} C_VEL
LIN {X 0,Y 580.043,Z 479.808,A -85,B 0,C 180,E1 -1887.222,E2 -1887.222} C_VEL
LIN {X 0,Y 580.039,Z 481.199,A -85,B 0,C 180,E1 -1887.917,E2 -1887.917} C_VEL
LIN {X 0,Y 580.04,Z 482.785,A -85,B 0,C 180,E1 -1889.306,E2 -1889.306} C_VEL
LIN {X 0,Y 580.037,Z 483,A -85,B 0,C 180,E1 -1890,E2 -1890} C_VEL
LIN {X 0,Y 580.046,Z 482.186,A -85,B 0,C 180,E1 -1891.389,E2 -1891.389} C_VEL
LIN {X 0,Y 580.039,Z 481.2,A -85,B 0,C 180,E1 -1892.083,E2 -1892.083} C_VEL
LIN {X 0,Y 580.043,Z 479.81,A -85,B 0,C 180,E1 -1892.778,E2 -1892.778} C_VEL
LIN {X 0,Y 580.11,Z 476.896,A -85,B 0,C 180,E1 -1893.821,E2 -1893.821} C_VEL
LIN {X 0,Y 580.053,Z 472.949,A -85,B 0,C 180,E1 -1894.865,E2 -1894.865} C_VEL
LIN {X 0,Y 580.139,Z 466.877,A -85,B 0,C 180,E1 -1896.085,E2 -1896.085} C_VEL
LIN {X 0,Y 580.184,Z 460.237,A -85,B 0,C 180,E1 -1897.132,E2 -1897.132} C_VEL
LIN {X 0,Y 580.25,Z 451.99,A -85,B 0,C 180,E1 -1898.182,E2 -1898.182} C_VEL
LIN {X 0,Y 580.308,Z 443.538,A -85,B 0,C 180,E1 -1899.058,E2 -1899.058} C_VEL
LIN {X 0,Y 580.419,Z 433.097,A -85,B 0,C 180,E1 -1899.936,E2 -1899.936} C_VEL
LIN {X 0,Y 580.512,Z 422.754,A -85,B 0,C 180,E1 -1900.639,E2 -1900.639} C_VEL
LIN {X 0,Y 580.581,Z 411.407,A -85,B 0,C 180,E1 -1901.256,E2 -1901.256} C_VEL
LIN {X 0,Y 580.654,Z 399.766,A -85,B 0,C 180,E1 -1901.741,E2 -1901.741} C_VEL
LIN {X 0,Y 580.729,Z 386.347,A -85,B 0,C 180,E1 -1902.138,E2 -1902.138} C_VEL
LIN {X 0,Y 580.79,Z 373.082,A -85,B 0,C 180,E1 -1902.381,E2 -1902.381} C_VEL
LIN {X 0,Y 580.787,Z 273.6,A -85,B 0,C 180,E1 -1903.618,E2 -1903.618} C_VEL
LIN {X 0,Y 580.389,Z 270.792,A -85,B 0,C 180,E1 -1903.68,E2 -1903.68} C_VEL
LIN {X 0,Y 580.536,Z 249.541,A -85,B 0,C 180,E1 -1906.709,E2 -1906.709} C_VEL
LIN {X 0,Y 580.704,Z 230.386,A -85,B 0,C 180,E1 -1909.479,E2 -1909.479} C_VEL
LIN {X 0,Y 580.908,Z 211.682,A -85,B 0,C 180,E1 -1912.214,E2 -1912.214} C_VEL
LIN {X 0,Y 580.272,Z 207.206,A -85,B 0,C 180,E1 -1912.923,E2 -1912.923} C_VEL
LIN {X 0,Y 580.29,Z 207.201,A -85,B 0,C 180,E1 -1915.081,E2 -1915.081} C_VEL
LIN {X 0,Y 580.291,Z 207.197,A -85,B 0,C 180,E1 -1918.186,E2 -1918.186} C_VEL
LIN {X 0,Y 580.273,Z 207.199,A -85,B 0,C 180,E1 -1920.692,E2 -1920.692} C_VEL
LIN {X 0,Y 580.304,Z 207.202,A -85,B 0,C 180,E1 -1923.316,E2 -1923.316} C_VEL
LIN {X 0,Y 580.244,Z 207.207,A -85,B 0,C 180,E1 -1925.756,E2 -1925.756} C_VEL
LIN {X 0,Y 580.285,Z 207.197,A -85,B 0,C 180,E1 -1928.147,E2 -1928.147} C_VEL
LIN {X 0,Y 580.295,Z 207.197,A -85,B 0,C 180,E1 -1930.844,E2 -1930.844} C_VEL
LIN {X 0,Y 580.27,Z 207.205,A -85,B 0,C 180,E1 -1933.659,E2 -1933.659} C_VEL
LIN {X 0,Y 580.244,Z 207.202,A -85,B 0,C 180,E1 -1936.613,E2 -1936.613} C_VEL
LIN {X 0,Y 580.294,Z 207.2,A -85,B 0,C 180,E1 -1939.156,E2 -1939.156} C_VEL
LIN {X 0,Y 580.284,Z 207.199,A -85,B 0,C 180,E1 -1941.928,E2 -1941.928} C_VEL
LIN {X 0,Y 580.234,Z 207.202,A -85,B 0,C 180,E1 -1944.451,E2 -1944.451} C_VEL
LIN {X 0,Y 580.289,Z 207.198,A -85,B 0,C 180,E1 -1946.975,E2 -1946.975} C_VEL
LIN {X 0,Y 580.293,Z 207.205,A -85,B 0,C 180,E1 -1949.425,E2 -1949.425} C_VEL
LIN {X 0,Y 580.258,Z 207.2,A -85,B 0,C 180,E1 -1952.149,E2 -1952.149} C_VEL
LIN {X 0,Y 580.3,Z 207.196,A -85,B 0,C 180,E1 -1954.92,E2 -1954.92} C_VEL
LIN {X 0,Y 580.268,Z 207.2,A -85,B 0,C 180,E1 -1957.947,E2 -1957.947} C_VEL
LIN {X 0,Y 580.297,Z 207.197,A -85,B 0,C 180,E1 -1960.913,E2 -1960.913} C_VEL
LIN {X 0,Y 580.267,Z 207.202,A -85,B 0,C 180,E1 -1963.825,E2 -1963.825} C_VEL
LIN {X 0,Y 580.324,Z 207.193,A -85,B 0,C 180,E1 -1965.983,E2 -1965.983} C_VEL
LIN {X 0,Y 580.307,Z 207.194,A -85,B 0,C 180,E1 -1968.827,E2 -1968.827} C_VEL
LIN {X 0,Y 580.327,Z 207.197,A -85,B 0,C 180,E1 -1971.644,E2 -1971.644} C_VEL
LIN {X 0,Y 580.284,Z 207.201,A -85,B 0,C 180,E1 -1973.742,E2 -1973.742} C_VEL
LIN {X 0,Y 580.272,Z 207.201,A -85,B 0,C 180,E1 -1975.833,E2 -1975.833} C_VEL
LIN {X 0,Y 580.344,Z 207.191,A -85,B 0,C 180,E1 -1977.918,E2 -1977.918} C_VEL
LIN {X 0,Y 580.346,Z 207.189,A -85,B 0,C 180,E1 -1980.694,E2 -1980.694} C_VEL
LIN {X 0,Y 580.279,Z 207.207,A -85,B 0,C 180,E1 -1983.472,E2 -1983.472} C_VEL
LIN {X 0,Y 580.326,Z 207.199,A -85,B 0,C 180,E1 -1985.56,E2 -1985.56} C_VEL
LIN {X 0,Y 580.309,Z 207.192,A -85,B 0,C 180,E1 -1988.356,E2 -1988.356} C_VEL
LIN {X 0,Y 580.302,Z 207.2,A -85,B 0,C 180,E1 -1991.191,E2 -1991.191} C_VEL
LIN {X 0,Y 580.316,Z 207.194,A -85,B 0,C 180,E1 -1994.017,E2 -1994.017} C_VEL
LIN {X 0,Y 580.291,Z 207.198,A -85,B 0,C 180,E1 -1996.906,E2 -1996.906} C_VEL
LIN {X 0,Y 580.283,Z 207.2,A -85,B 0,C 180,E1 -1999.823,E2 -1999.823} C_VEL
LIN {X 0,Y 580.285,Z 207.205,A -85,B 0,C 180,E1 -2001.305,E2 -2001.305} C_VEL
LIN {X 0,Y 579.577,Z 207.3,A -85,B 0,C 180,E1 -2001.884,E2 -2001.884} C_VEL
LIN {X 0,Y 576.7,Z 207.656,A -85,B 0,C 180,E1 -2002.824,E2 -2002.824} C_VEL
LIN {X 0,Y 574.305,Z 207.949,A -85,B 0,C 180,E1 -2003.58,E2 -2003.58} C_VEL
LIN {X 0,Y 573.294,Z 208.068,A -85,B 0,C 180,E1 -2004.164,E2 -2004.164} C_VEL
LIN {X 0,Y 573.221,Z 208.076,A -85,B 0,C 180,E1 -2004.362,E2 -2004.362} C_VEL
LIN {X 0,Y 573.21,Z 208.08,A -85,B 0,C 180,E1 -2006.978,E2 -2006.978} C_VEL
LIN {X 0,Y 573.239,Z 208.083,A -85,B 0,C 180,E1 -2009.487,E2 -2009.487} C_VEL
LIN {X 0,Y 573.253,Z 208.073,A -85,B 0,C 180,E1 -2012.645,E2 -2012.645} C_VEL
LIN {X 0,Y 573.205,Z 208.085,A -85,B 0,C 180,E1 -2015.188,E2 -2015.188} C_VEL
LIN {X 0,Y 573.232,Z 208.079,A -85,B 0,C 180,E1 -2017.808,E2 -2017.808} C_VEL
LIN {X 0,Y 573.247,Z 208.073,A -85,B 0,C 180,E1 -2020.525,E2 -2020.525} C_VEL
LIN {X 0,Y 573.232,Z 208.085,A -85,B 0,C 180,E1 -2023.36,E2 -2023.36} C_VEL
LIN {X 0,Y 573.212,Z 208.077,A -85,B 0,C 180,E1 -2026.335,E2 -2026.335} C_VEL
LIN {X 0,Y 573.228,Z 208.076,A -85,B 0,C 180,E1 -2028.543,E2 -2028.543} C_VEL
LIN {X 0,Y 573.241,Z 208.083,A -85,B 0,C 180,E1 -2031.298,E2 -2031.298} C_VEL
LIN {X 0,Y 573.196,Z 208.082,A -85,B 0,C 180,E1 -2034.021,E2 -2034.021} C_VEL
LIN {X 0,Y 573.244,Z 208.074,A -85,B 0,C 180,E1 -2036.516,E2 -2036.516} C_VEL
LIN {X 0,Y 573.229,Z 208.081,A -85,B 0,C 180,E1 -2039.118,E2 -2039.118} C_VEL
LIN {X 0,Y 573.23,Z 208.084,A -85,B 0,C 180,E1 -2041.435,E2 -2041.435} C_VEL
LIN {X 0,Y 573.279,Z 208.217,A -85,B 0,C 180,E1 -2044.299,E2 -2044.299} C_VEL
LIN {X 0,Y 573.506,Z 214.353,A -85,B 0,C 180,E1 -2045.377,E2 -2045.377} C_VEL
LIN {X 0,Y 573.372,Z 229.599,A -85,B 0,C 180,E1 -2048.047,E2 -2048.047} C_VEL
LIN {X 0,Y 573.291,Z 242.13,A -85,B 0,C 180,E1 -2050.216,E2 -2050.216} C_VEL
LIN {X 0,Y 574.039,Z 248.749,A -85,B 0,C 180,E1 -2050.329,E2 -2050.329} C_VEL
LIN {X 0,Y 573.823,Z 349.717,A -85,B 0,C 180,E1 -2051.616,E2 -2051.616} C_VEL
LIN {X 0,Y 573.749,Z 363.005,A -85,B 0,C 180,E1 -2051.937,E2 -2051.937} C_VEL
LIN {X 0,Y 573.69,Z 375.115,A -85,B 0,C 180,E1 -2052.368,E2 -2052.368} C_VEL
LIN {X 0,Y 573.588,Z 386.274,A -85,B 0,C 180,E1 -2052.899,E2 -2052.899} C_VEL
LIN {X 0,Y 573.448,Z 398.159,A -85,B 0,C 180,E1 -2053.627,E2 -2053.627} C_VEL
LIN {X 0,Y 573.332,Z 408.784,A -85,B 0,C 180,E1 -2054.446,E2 -2054.446} C_VEL
LIN {X 0,Y 573.242,Z 417.42,A -85,B 0,C 180,E1 -2055.26,E2 -2055.26} C_VEL
LIN {X 0,Y 573.154,Z 426.745,A -85,B 0,C 180,E1 -2056.347,E2 -2056.347} C_VEL
LIN {X 0,Y 573.097,Z 434.198,A -85,B 0,C 180,E1 -2057.428,E2 -2057.428} C_VEL
LIN {X 0,Y 573.041,Z 439.221,A -85,B 0,C 180,E1 -2058.325,E2 -2058.325} C_VEL
LIN {X 0,Y 573.017,Z 444.074,A -85,B 0,C 180,E1 -2059.399,E2 -2059.399} C_VEL
LIN {X 0,Y 572.987,Z 447.778,A -85,B 0,C 180,E1 -2060.469,E2 -2060.469} C_VEL
LIN {X 0,Y 572.956,Z 450.443,A -85,B 0,C 180,E1 -2061.536,E2 -2061.536} C_VEL
LIN {X 0,Y 572.978,Z 451.689,A -85,B 0,C 180,E1 -2062.246,E2 -2062.246} C_VEL
LIN {X 0,Y 573.011,Z 452.856,A -85,B 0,C 180,E1 -2063.45,E2 -2063.45} C_VEL
LIN {X 0,Y 572.991,Z 452.934,A -85,B 0,C 180,E1 -2064.369,E2 -2064.369} C_VEL
LIN {X 0,Y 572.936,Z 452.565,A -85,B 0,C 180,E1 -2065.074,E2 -2065.074} C_VEL
LIN {X 0,Y 573.007,Z 451.788,A -85,B 0,C 180,E1 -2065.78,E2 -2065.78} C_VEL
LIN {X 0,Y 573.007,Z 450.584,A -85,B 0,C 180,E1 -2066.484,E2 -2066.484} C_VEL
LIN {X 0,Y 573.012,Z 448.021,A -85,B 0,C 180,E1 -2067.54,E2 -2067.54} C_VEL
LIN {X 0,Y 572.971,Z 444.468,A -85,B 0,C 180,E1 -2068.594,E2 -2068.594} C_VEL
LIN {X 0,Y 573.054,Z 439.818,A -85,B 0,C 180,E1 -2069.649,E2 -2069.649} C_VEL
LIN {X 0,Y 573.105,Z 432.834,A -85,B 0,C 180,E1 -2070.878,E2 -2070.878} C_VEL
LIN {X 0,Y 573.217,Z 425.289,A -85,B 0,C 180,E1 -2071.932,E2 -2071.932} C_VEL
LIN {X 0,Y 573.257,Z 415.848,A -85,B 0,C 180,E1 -2072.987,E2 -2072.987} C_VEL
LIN {X 0,Y 573.383,Z 406.126,A -85,B 0,C 180,E1 -2073.865,E2 -2073.865} C_VEL
LIN {X 0,Y 573.485,Z 395.282,A -85,B 0,C 180,E1 -2074.657,E2 -2074.657} C_VEL
LIN {X 0,Y 573.629,Z 382.967,A -85,B 0,C 180,E1 -2075.36,E2 -2075.36} C_VEL
LIN {X 0,Y 573.698,Z 370.911,A -85,B 0,C 180,E1 -2075.889,E2 -2075.889} C_VEL
LIN {X 0,Y 573.841,Z 358.273,A -85,B 0,C 180,E1 -2076.284,E2 -2076.284} C_VEL
LIN {X 0,Y 573.892,Z 345.459,A -85,B 0,C 180,E1 -2076.542,E2 -2076.542} C_VEL
LIN {X 0,Y 573.976,Z 246.559,A -85,B 0,C 180,E1 -2077.79,E2 -2077.79} C_VEL
LIN {X 0,Y 573.282,Z 242.077,A -85,B 0,C 180,E1 -2077.883,E2 -2077.883} C_VEL
LIN {X 0,Y 573.432,Z 225.412,A -85,B 0,C 180,E1 -2080.772,E2 -2080.772} C_VEL
LIN {X 0,Y 573.539,Z 210.073,A -85,B 0,C 180,E1 -2083.463,E2 -2083.463} C_VEL
LIN {X 0,Y 573.274,Z 208.076,A -85,B 0,C 180,E1 -2083.831,E2 -2083.831} C_VEL
LIN {X 0,Y 573.263,Z 208.076,A -85,B 0,C 180,E1 -2087.111,E2 -2087.111} C_VEL
LIN {X 0,Y 573.244,Z 208.075,A -85,B 0,C 180,E1 -2090.077,E2 -2090.077} C_VEL
LIN {X 0,Y 573.236,Z 208.079,A -85,B 0,C 180,E1 -2092.338,E2 -2092.338} C_VEL
LIN {X 0,Y 573.246,Z 208.074,A -85,B 0,C 180,E1 -2095.41,E2 -2095.41} C_VEL
LIN {X 0,Y 573.23,Z 208.083,A -85,B 0,C 180,E1 -2098.565,E2 -2098.565} C_VEL
LIN {X 0,Y 573.226,Z 208.08,A -85,B 0,C 180,E1 -2100.993,E2 -2100.993} C_VEL
LIN {X 0,Y 573.266,Z 208.071,A -85,B 0,C 180,E1 -2103.524,E2 -2103.524} C_VEL
LIN {X 0,Y 573.196,Z 208.081,A -85,B 0,C 180,E1 -2106.053,E2 -2106.053} C_VEL
LIN {X 0,Y 573.242,Z 208.084,A -85,B 0,C 180,E1 -2108.702,E2 -2108.702} C_VEL
LIN {X 0,Y 573.23,Z 208.075,A -85,B 0,C 180,E1 -2111.592,E2 -2111.592} C_VEL
LIN {X 0,Y 573.231,Z 208.08,A -85,B 0,C 180,E1 -2114.334,E2 -2114.334} C_VEL
LIN {X 0,Y 573.235,Z 208.075,A -85,B 0,C 180,E1 -2117.359,E2 -2117.359} C_VEL
LIN {X 0,Y 573.239,Z 208.08,A -85,B 0,C 180,E1 -2120.392,E2 -2120.392} C_VEL
LIN {X 0,Y 573.233,Z 208.078,A -85,B 0,C 180,E1 -2123.076,E2 -2123.076} C_VEL
LIN {X 0,Y 573.265,Z 208.07,A -85,B 0,C 180,E1 -2125.671,E2 -2125.671} C_VEL
LIN {X 0,Y 573.239,Z 208.077,A -85,B 0,C 180,E1 -2128.184,E2 -2128.184} C_VEL
LIN {X 0,Y 573.261,Z 208.082,A -85,B 0,C 180,E1 -2130.634,E2 -2130.634} C_VEL
LIN {X 0,Y 573.21,Z 208.081,A -85,B 0,C 180,E1 -2133.022,E2 -2133.022} C_VEL
LIN {X 0,Y 573.237,Z 208.075,A -85,B 0,C 180,E1 -2135.364,E2 -2135.364} C_VEL
LIN {X 0,Y 573.232,Z 208.075,A -85,B 0,C 180,E1 -2137.662,E2 -2137.662} C_VEL
LIN {X 0,Y 573.267,Z 208.08,A -85,B 0,C 180,E1 -2140.67,E2 -2140.67} C_VEL
LIN {X 0,Y 573.239,Z 208.074,A -85,B 0,C 180,E1 -2143.621,E2 -2143.621} C_VEL
LIN {X 0,Y 573.26,Z 208.071,A -85,B 0,C 180,E1 -2145.807,E2 -2145.807} C_VEL
LIN {X 0,Y 573.264,Z 208.079,A -85,B 0,C 180,E1 -2148.745,E2 -2148.745} C_VEL
LIN {X 0,Y 573.254,Z 208.072,A -85,B 0,C 180,E1 -2151.54,E2 -2151.54} C_VEL
LIN {X 0,Y 573.294,Z 208.073,A -85,B 0,C 180,E1 -2154.372,E2 -2154.372} C_VEL
LIN {X 0,Y 573.311,Z 208.066,A -85,B 0,C 180,E1 -2157.892,E2 -2157.892} C_VEL
LIN {X 0,Y 573.332,Z 208.071,A -85,B 0,C 180,E1 -2160.702,E2 -2160.702} C_VEL
LIN {X 0,Y 573.304,Z 208.072,A -85,B 0,C 180,E1 -2162.811,E2 -2162.811} C_VEL
LIN {X 0,Y 573.28,Z 208.069,A -85,B 0,C 180,E1 -2165.628,E2 -2165.628} C_VEL
LIN {X 0,Y 573.268,Z 208.07,A -85,B 0,C 180,E1 -2167.75,E2 -2167.75} C_VEL
LIN {X 0,Y 573.266,Z 208.081,A -85,B 0,C 180,E1 -2170.597,E2 -2170.597} C_VEL
LIN {X 0,Y 573.262,Z 208.079,A -85,B 0,C 180,E1 -2172.749,E2 -2172.749} C_VEL
LIN {X 0,Y 573.232,Z 208.079,A -85,B 0,C 180,E1 -2174.92,E2 -2174.92} C_VEL
LIN {X 0,Y 573.231,Z 208.076,A -85,B 0,C 180,E1 -2177.849,E2 -2177.849} C_VEL
LIN {X 0,Y 573.241,Z 208.076,A -85,B 0,C 180,E1 -2180.077,E2 -2180.077} C_VEL
LIN {X 0,Y 573.232,Z 208.081,A -85,B 0,C 180,E1 -2182.338,E2 -2182.338} C_VEL
LIN {X 0,Y 573.243,Z 208.073,A -85,B 0,C 180,E1 -2185.411,E2 -2185.411} C_VEL
LIN {X 0,Y 573.228,Z 208.086,A -85,B 0,C 180,E1 -2188.565,E2 -2188.565} C_VEL
LIN {X 0,Y 573.223,Z 208.079,A -85,B 0,C 180,E1 -2190.994,E2 -2190.994} C_VEL
LIN {X 0,Y 573.242,Z 208.073,A -85,B 0,C 180,E1 -2193.521,E2 -2193.521} C_VEL
LIN {X 0,Y 573.193,Z 208.082,A -85,B 0,C 180,E1 -2196.053,E2 -2196.053} C_VEL
LIN {X 0,Y 573.239,Z 208.082,A -85,B 0,C 180,E1 -2198.702,E2 -2198.702} C_VEL
LIN {X 0,Y 573.227,Z 208.075,A -85,B 0,C 180,E1 -2201.593,E2 -2201.593} C_VEL
LIN {X 0,Y 573.217,Z 208.083,A -85,B 0,C 180,E1 -2204.335,E2 -2204.335} C_VEL
LIN {X 0,Y 573.233,Z 208.075,A -85,B 0,C 180,E1 -2207.36,E2 -2207.36} C_VEL
LIN {X 0,Y 573.237,Z 208.082,A -85,B 0,C 180,E1 -2210.392,E2 -2210.392} C_VEL
LIN {X 0,Y 573.231,Z 208.077,A -85,B 0,C 180,E1 -2213.076,E2 -2213.076} C_VEL
LIN {X 0,Y 573.264,Z 208.071,A -85,B 0,C 180,E1 -2215.671,E2 -2215.671} C_VEL
LIN {X 0,Y 573.237,Z 208.079,A -85,B 0,C 180,E1 -2218.184,E2 -2218.184} C_VEL
LIN {X 0,Y 573.257,Z 208.081,A -85,B 0,C 180,E1 -2220.634,E2 -2220.634} C_VEL
LIN {X 0,Y 573.209,Z 208.081,A -85,B 0,C 180,E1 -2223.022,E2 -2223.022} C_VEL
LIN {X 0,Y 573.237,Z 208.075,A -85,B 0,C 180,E1 -2225.364,E2 -2225.364} C_VEL
LIN {X 0,Y 573.256,Z 208.287,A -85,B 0,C 180,E1 -2226.997,E2 -2226.997} C_VEL
LIN {X 0,Y 573.956,Z 212.77,A -85,B 0,C 180,E1 -2227.692,E2 -2227.692} C_VEL
LIN {X 0,Y 573.784,Z 230.644,A -85,B 0,C 180,E1 -2230.316,E2 -2230.316} C_VEL
LIN {X 0,Y 573.542,Z 249.142,A -85,B 0,C 180,E1 -2233.023,E2 -2233.023} C_VEL
LIN {X 0,Y 573.402,Z 270.792,A -85,B 0,C 180,E1 -2236.15,E2 -2236.15} C_VEL
LIN {X 0,Y 574.062,Z 276.51,A -85,B 0,C 180,E1 -2236.256,E2 -2236.256} C_VEL
LIN {X 0,Y 573.845,Z 378.947,A -85,B 0,C 180,E1 -2237.557,E2 -2237.557} C_VEL
LIN {X 0,Y 573.785,Z 392.219,A -85,B 0,C 180,E1 -2237.87,E2 -2237.87} C_VEL
LIN {X 0,Y 573.676,Z 404.376,A -85,B 0,C 180,E1 -2238.294,E2 -2238.294} C_VEL
LIN {X 0,Y 573.57,Z 416.764,A -85,B 0,C 180,E1 -2238.881,E2 -2238.881} C_VEL
LIN {X 0,Y 573.44,Z 428.2,A -85,B 0,C 180,E1 -2239.585,E2 -2239.585} C_VEL
LIN {X 0,Y 573.331,Z 438.602,A -85,B 0,C 180,E1 -2240.386,E2 -2240.386} C_VEL
LIN {X 0,Y 573.241,Z 447.113,A -85,B 0,C 180,E1 -2241.185,E2 -2241.185} C_VEL
LIN {X 0,Y 573.161,Z 454.961,A -85,B 0,C 180,E1 -2242.071,E2 -2242.071} C_VEL
LIN {X 0,Y 573.072,Z 462.955,A -85,B 0,C 180,E1 -2243.185,E2 -2243.185} C_VEL
LIN {X 0,Y 573.07,Z 469.68,A -85,B 0,C 180,E1 -2244.37,E2 -2244.37} C_VEL
LIN {X 0,Y 573.028,Z 474.372,A -85,B 0,C 180,E1 -2245.428,E2 -2245.428} C_VEL
LIN {X 0,Y 573.022,Z 477.958,A -85,B 0,C 180,E1 -2246.484,E2 -2246.484} C_VEL
LIN {X 0,Y 572.959,Z 479.808,A -85,B 0,C 180,E1 -2247.188,E2 -2247.188} C_VEL
LIN {X 0,Y 572.946,Z 482.185,A -85,B 0,C 180,E1 -2248.594,E2 -2248.594} C_VEL
LIN {X 0,Y 572.938,Z 483,A -85,B 0,C 180,E1 -2250,E2 -2250} C_VEL
LIN {X 0,Y 572.946,Z 482.186,A -85,B 0,C 180,E1 -2251.406,E2 -2251.406} C_VEL
LIN {X 0,Y 572.939,Z 481.199,A -85,B 0,C 180,E1 -2252.109,E2 -2252.109} C_VEL
LIN {X 0,Y 572.959,Z 479.81,A -85,B 0,C 180,E1 -2252.812,E2 -2252.812} C_VEL
LIN {X 0,Y 573.015,Z 476.896,A -85,B 0,C 180,E1 -2253.868,E2 -2253.868} C_VEL
LIN {X 0,Y 572.963,Z 472.949,A -85,B 0,C 180,E1 -2254.926,E2 -2254.926} C_VEL
LIN {X 0,Y 573.064,Z 466.876,A -85,B 0,C 180,E1 -2256.16,E2 -2256.16} C_VEL
LIN {X 0,Y 573.119,Z 460.237,A -85,B 0,C 180,E1 -2257.221,E2 -2257.221} C_VEL
LIN {X 0,Y 573.201,Z 451.991,A -85,B 0,C 180,E1 -2258.283,E2 -2258.283} C_VEL
LIN {X 0,Y 573.287,Z 443.538,A -85,B 0,C 180,E1 -2259.17,E2 -2259.17} C_VEL
LIN {X 0,Y 573.424,Z 433.096,A -85,B 0,C 180,E1 -2260.058,E2 -2260.058} C_VEL
LIN {X 0,Y 573.555,Z 421.4,A -85,B 0,C 180,E1 -2260.855,E2 -2260.855} C_VEL
